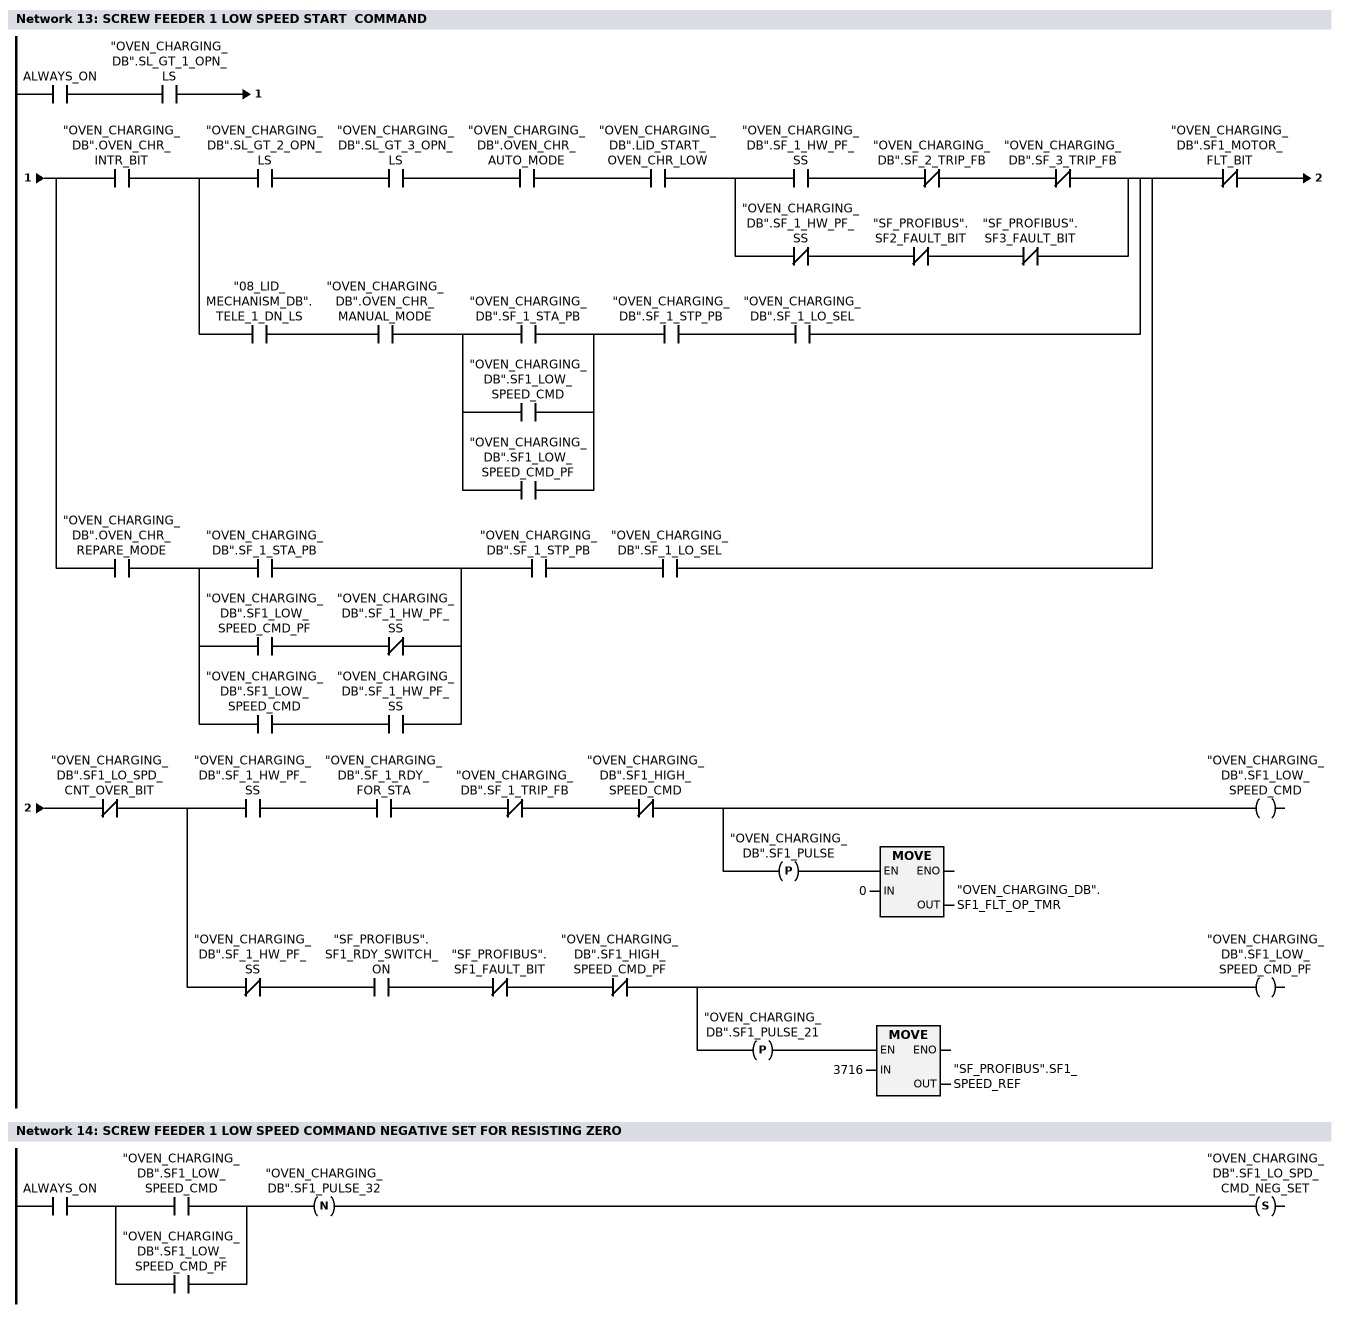
[picture p96: OVEN_CHARGING_SF networks 13-14]
NETWORK
TITLE = SCREW FEEDER 1 LOW SPEED START  COMMAND
      A     "ALWAYS_ON";
      A     "OVEN_CHARGING_DB".SL_GT_1_OPN_LS;
      A(;
      A     "OVEN_CHARGING_DB".OVEN_CHR_INTR_BIT;
      A(;
      A     "OVEN_CHARGING_DB".SL_GT_2_OPN_LS;
      A     "OVEN_CHARGING_DB".SL_GT_3_OPN_LS;
      A     "OVEN_CHARGING_DB".OVEN_CHR_AUTO_MODE;
      A     "OVEN_CHARGING_DB".LID_START_OVEN_CHR_LOW;
      A(;
      A     "OVEN_CHARGING_DB".SF_1_HW_PF_SS;
      AN    "OVEN_CHARGING_DB".SF_2_TRIP_FB;
      AN    "OVEN_CHARGING_DB".SF_3_TRIP_FB;
      O;
      AN    "OVEN_CHARGING_DB".SF_1_HW_PF_SS;
      AN    "SF_PROFIBUS".SF2_FAULT_BIT;
      AN    "SF_PROFIBUS".SF3_FAULT_BIT;
      );
      O;
      A     "08_LID_MECHANISM_DB".TELE_1_DN_LS;
      A     "OVEN_CHARGING_DB".OVEN_CHR_MANUAL_MODE;
      A(;
      O     "OVEN_CHARGING_DB".SF_1_STA_PB;
      O     "OVEN_CHARGING_DB".SF1_LOW_SPEED_CMD;
      O     "OVEN_CHARGING_DB".SF1_LOW_SPEED_CMD_PF;
      );
      A     "OVEN_CHARGING_DB".SF_1_STP_PB;
      A     "OVEN_CHARGING_DB".SF_1_LO_SEL;
      );
      O;
      A     "OVEN_CHARGING_DB".OVEN_CHR_REPARE_MODE;
      A(;
      O     "OVEN_CHARGING_DB".SF_1_STA_PB;
      O;
      A     "OVEN_CHARGING_DB".SF1_LOW_SPEED_CMD_PF;
      AN    "OVEN_CHARGING_DB".SF_1_HW_PF_SS;
      O;
      A     "OVEN_CHARGING_DB".SF1_LOW_SPEED_CMD;
      A     "OVEN_CHARGING_DB".SF_1_HW_PF_SS;
      );
      A     "OVEN_CHARGING_DB".SF_1_STP_PB;
      A     "OVEN_CHARGING_DB".SF_1_LO_SEL;
      );
      AN    "OVEN_CHARGING_DB".SF1_MOTOR_FLT_BIT;
      AN    "OVEN_CHARGING_DB".SF1_LO_SPD_CNT_OVER_BIT;
      =     L 0.0;
      A     L 0.0;
      A     "OVEN_CHARGING_DB".SF_1_HW_PF_SS;
      A     "OVEN_CHARGING_DB".SF_1_RDY_FOR_STA;
      AN    "OVEN_CHARGING_DB".SF_1_TRIP_FB;
      AN    "OVEN_CHARGING_DB".SF1_HIGH_SPEED_CMD;
      =     L 0.1;
      A     L 0.1;
      BLD   102;
      =     "OVEN_CHARGING_DB".SF1_LOW_SPEED_CMD;
      A     L 0.1;
      FP    "OVEN_CHARGING_DB".SF1_PULSE;
      JNB   _007;
      L     0;
      T     "OVEN_CHARGING_DB".SF1_FLT_OP_TMR;
_007: NOP   0;
      A     L 0.0;
      AN    "OVEN_CHARGING_DB".SF_1_HW_PF_SS;
      A     "SF_PROFIBUS".SF1_RDY_SWITCH_ON;
      AN    "SF_PROFIBUS".SF1_FAULT_BIT;
      AN    "OVEN_CHARGING_DB".SF1_HIGH_SPEED_CMD_PF;
      =     L 0.1;
      A     L 0.1;
      BLD   102;
      =     "OVEN_CHARGING_DB".SF1_LOW_SPEED_CMD_PF;
      A     L 0.1;
      FP    "OVEN_CHARGING_DB".SF1_PULSE_21;
      JNB   _008;
      L     3716;
      T     "SF_PROFIBUS".SF1_SPEED_REF;
_008: NOP   0;
NETWORK
TITLE = SCREW FEEDER 1 LOW SPEED COMMAND NEGATIVE SET FOR RESISTING ZERO
      A     "ALWAYS_ON";
      A(;
      O     "OVEN_CHARGING_DB".SF1_LOW_SPEED_CMD;
      O     "OVEN_CHARGING_DB".SF1_LOW_SPEED_CMD_PF;
      );
      FN    "OVEN_CHARGING_DB".SF1_PULSE_32;
      S     "OVEN_CHARGING_DB".SF1_LO_SPD_CMD_NEG_SET;
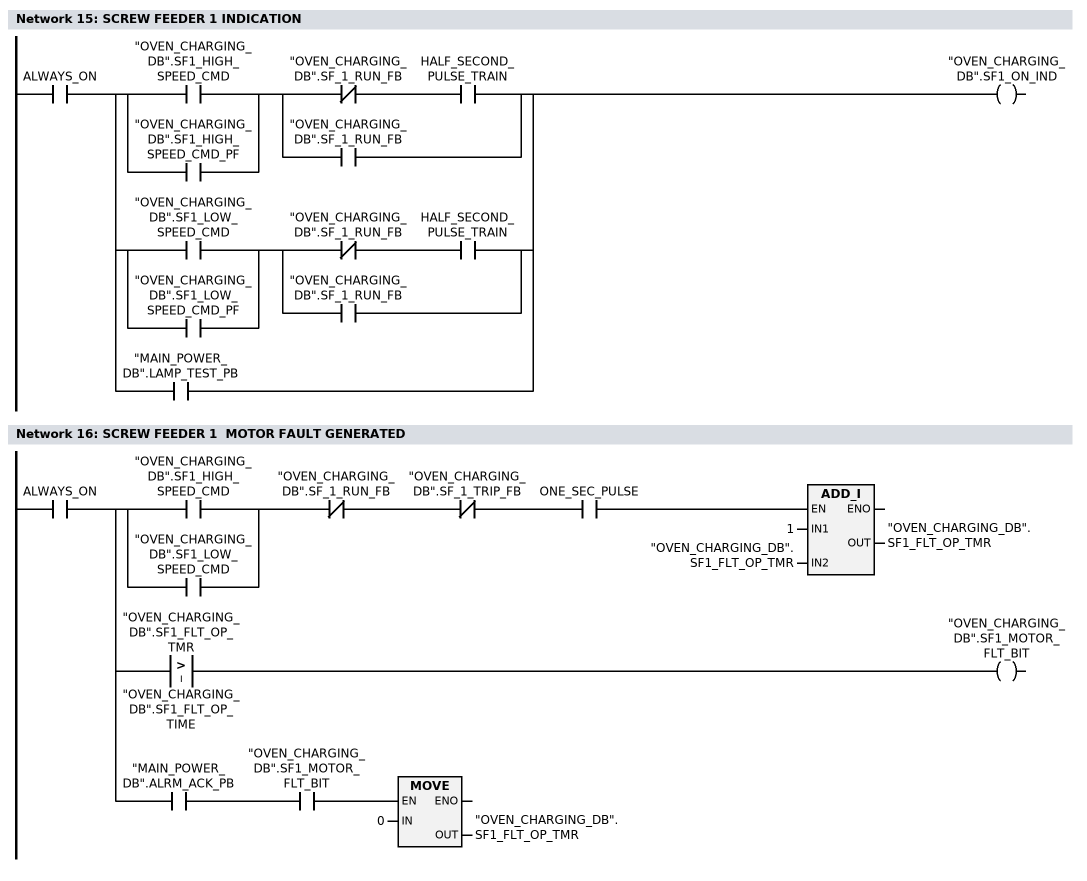
NETWORK
TITLE = SCREW FEEDER 1 INDICATION
      A     "ALWAYS_ON";
      A(;
      A(;
      O     "OVEN_CHARGING_DB".SF1_HIGH_SPEED_CMD;
      O     "OVEN_CHARGING_DB".SF1_HIGH_SPEED_CMD_PF;
      );
      A(;
      AN    "OVEN_CHARGING_DB".SF_1_RUN_FB;
      A     "HALF_SECOND_PULSE_TRAIN";
      O     "OVEN_CHARGING_DB".SF_1_RUN_FB;
      );
      O;
      A(;
      O     "OVEN_CHARGING_DB".SF1_LOW_SPEED_CMD;
      O     "OVEN_CHARGING_DB".SF1_LOW_SPEED_CMD_PF;
      );
      A(;
      AN    "OVEN_CHARGING_DB".SF_1_RUN_FB;
      A     "HALF_SECOND_PULSE_TRAIN";
      O     "OVEN_CHARGING_DB".SF_1_RUN_FB;
      );
      O     "MAIN_POWER_DB".LAMP_TEST_PB;
      );
      =     "OVEN_CHARGING_DB".SF1_ON_IND;
NETWORK
TITLE = SCREW FEEDER 1  MOTOR FAULT GENERATED
      A     "ALWAYS_ON";
      =     L 0.0;
      A     L 0.0;
      A(;
      O     "OVEN_CHARGING_DB".SF1_HIGH_SPEED_CMD;
      O     "OVEN_CHARGING_DB".SF1_LOW_SPEED_CMD;
      );
      AN    "OVEN_CHARGING_DB".SF_1_RUN_FB;
      AN    "OVEN_CHARGING_DB".SF_1_TRIP_FB;
      A     "ONE_SEC_PULSE";
      JNB   _009;
      L     1;
      L     "OVEN_CHARGING_DB".SF1_FLT_OP_TMR;
      +I;
      T     "OVEN_CHARGING_DB".SF1_FLT_OP_TMR;
_009: NOP   0;
      A     L 0.0;
      A(;
      L     "OVEN_CHARGING_DB".SF1_FLT_OP_TMR;
      L     "OVEN_CHARGING_DB".SF1_FLT_OP_TIME;
      >I;
      );
      =     "OVEN_CHARGING_DB".SF1_MOTOR_FLT_BIT;
      A     L 0.0;
      A     "MAIN_POWER_DB".ALRM_ACK_PB;
      A     "OVEN_CHARGING_DB".SF1_MOTOR_FLT_BIT;
      JNB   _00a;
      L     0;
      T     "OVEN_CHARGING_DB".SF1_FLT_OP_TMR;
_00a: NOP   0;
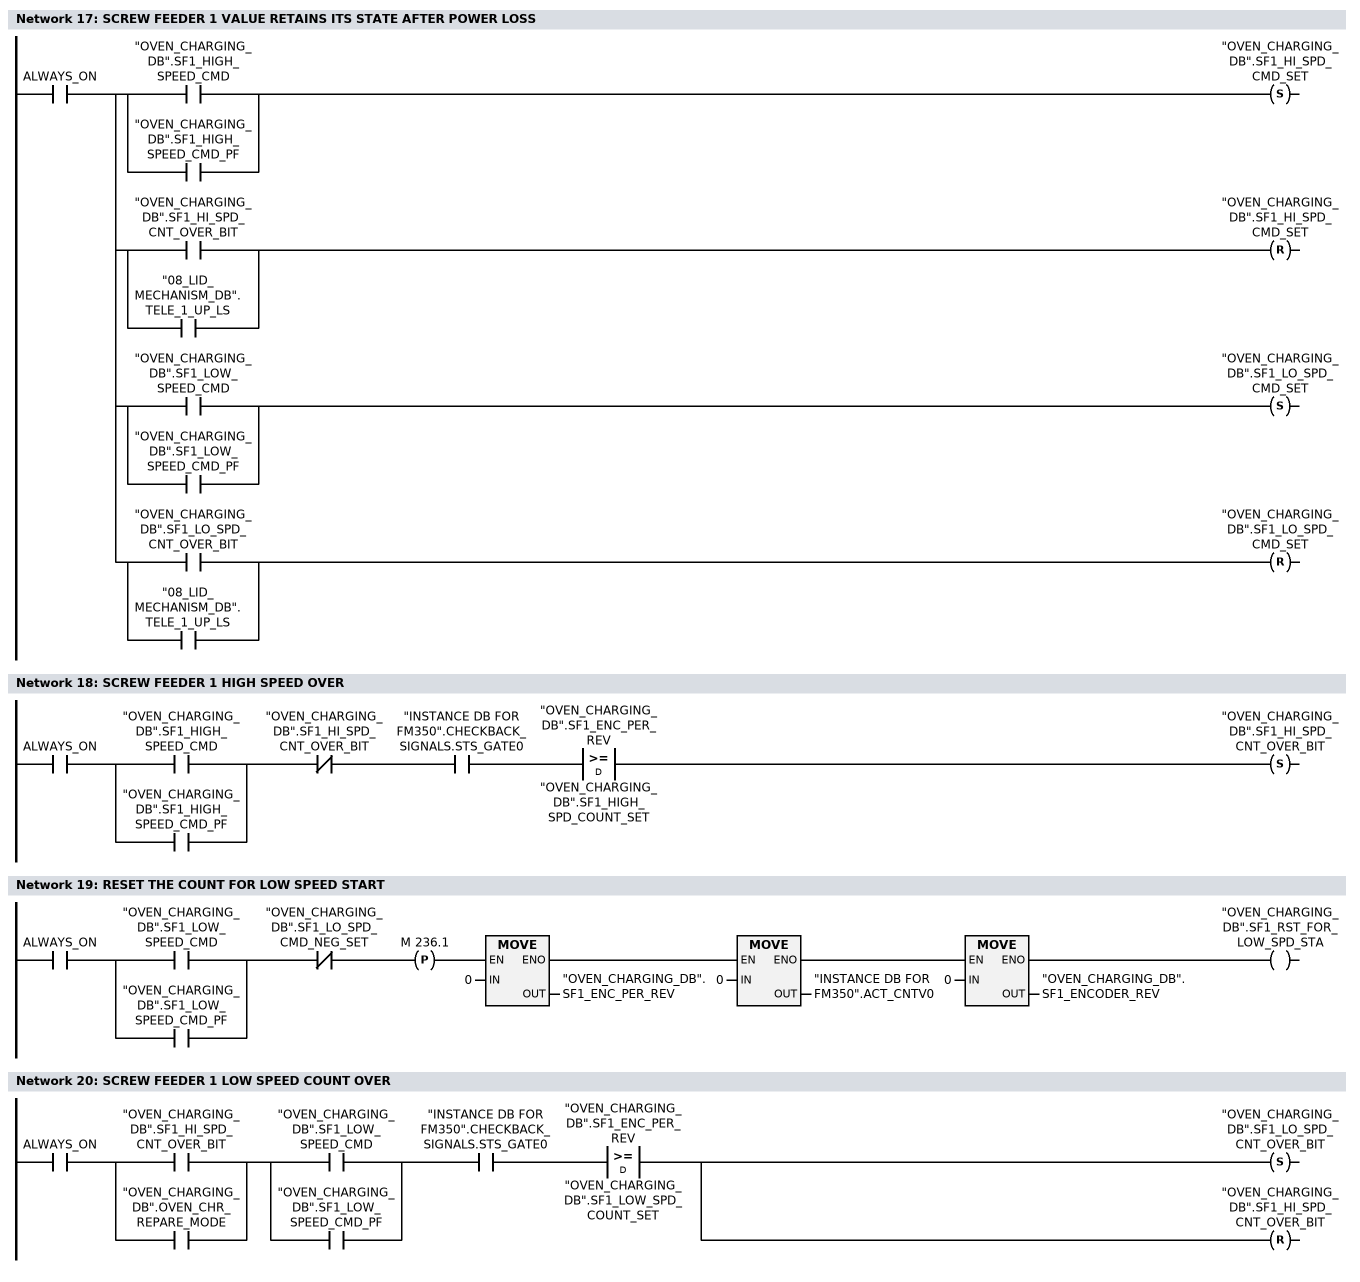
NETWORK
TITLE = SCREW FEEDER 1 VALUE RETAINS ITS STATE AFTER POWER LOSS
      A     "ALWAYS_ON";
      =     L 0.0;
      A     L 0.0;
      A(;
      O     "OVEN_CHARGING_DB".SF1_HIGH_SPEED_CMD;
      O     "OVEN_CHARGING_DB".SF1_HIGH_SPEED_CMD_PF;
      );
      S     "OVEN_CHARGING_DB".SF1_HI_SPD_CMD_SET;
      A     L 0.0;
      A(;
      O     "OVEN_CHARGING_DB".SF1_HI_SPD_CNT_OVER_BIT;
      O     "08_LID_MECHANISM_DB".TELE_1_UP_LS;
      );
      R     "OVEN_CHARGING_DB".SF1_HI_SPD_CMD_SET;
      A     L 0.0;
      A(;
      O     "OVEN_CHARGING_DB".SF1_LOW_SPEED_CMD;
      O     "OVEN_CHARGING_DB".SF1_LOW_SPEED_CMD_PF;
      );
      S     "OVEN_CHARGING_DB".SF1_LO_SPD_CMD_SET;
      A     L 0.0;
      A(;
      O     "OVEN_CHARGING_DB".SF1_LO_SPD_CNT_OVER_BIT;
      O     "08_LID_MECHANISM_DB".TELE_1_UP_LS;
      );
      R     "OVEN_CHARGING_DB".SF1_LO_SPD_CMD_SET;
NETWORK
TITLE = SCREW FEEDER 1 HIGH SPEED OVER
      A     "ALWAYS_ON";
      A(;
      O     "OVEN_CHARGING_DB".SF1_HIGH_SPEED_CMD;
      O     "OVEN_CHARGING_DB".SF1_HIGH_SPEED_CMD_PF;
      );
      AN    "OVEN_CHARGING_DB".SF1_HI_SPD_CNT_OVER_BIT;
      A     "INSTANCE DB FOR FM350".CHECKBACK_SIGNALS.STS_GATE0;
      A(;
      L     "OVEN_CHARGING_DB".SF1_ENC_PER_REV;
      L     "OVEN_CHARGING_DB".SF1_HIGH_SPD_COUNT_SET;
      >=D;
      );
      S     "OVEN_CHARGING_DB".SF1_HI_SPD_CNT_OVER_BIT;
NETWORK
TITLE = RESET THE COUNT FOR LOW SPEED START
      A(;
      A(;
      A     "ALWAYS_ON";
      A(;
      O     "OVEN_CHARGING_DB".SF1_LOW_SPEED_CMD;
      O     "OVEN_CHARGING_DB".SF1_LOW_SPEED_CMD_PF;
      );
      AN    "OVEN_CHARGING_DB".SF1_LO_SPD_CMD_NEG_SET;
      FP    M 236.1;
      JNB   _00b;
      L     0;
      T     "OVEN_CHARGING_DB".SF1_ENC_PER_REV;
      SET;
      SAVE;
      CLR;
_00b: A     BR;
      );
      JNB   _00c;
      L     0;
      T     "INSTANCE DB FOR FM350".ACT_CNTV0;
      SET;
      SAVE;
      CLR;
_00c: A     BR;
      );
      JNB   _00d;
      L     0;
      T     "OVEN_CHARGING_DB".SF1_ENCODER_REV;
      SET;
      SAVE;
      CLR;
_00d: A     BR;
      =     "OVEN_CHARGING_DB".SF1_RST_FOR_LOW_SPD_STA;
NETWORK
TITLE = SCREW FEEDER 1 LOW SPEED COUNT OVER
      A     "ALWAYS_ON";
      A(;
      O     "OVEN_CHARGING_DB".SF1_HI_SPD_CNT_OVER_BIT;
      O     "OVEN_CHARGING_DB".OVEN_CHR_REPARE_MODE;
      );
      A(;
      O     "OVEN_CHARGING_DB".SF1_LOW_SPEED_CMD;
      O     "OVEN_CHARGING_DB".SF1_LOW_SPEED_CMD_PF;
      );
      A     "INSTANCE DB FOR FM350".CHECKBACK_SIGNALS.STS_GATE0;
      A(;
      L     "OVEN_CHARGING_DB".SF1_ENC_PER_REV;
      L     "OVEN_CHARGING_DB".SF1_LOW_SPD_COUNT_SET;
      >=D;
      );
      S     "OVEN_CHARGING_DB".SF1_LO_SPD_CNT_OVER_BIT;
      R     "OVEN_CHARGING_DB".SF1_HI_SPD_CNT_OVER_BIT;
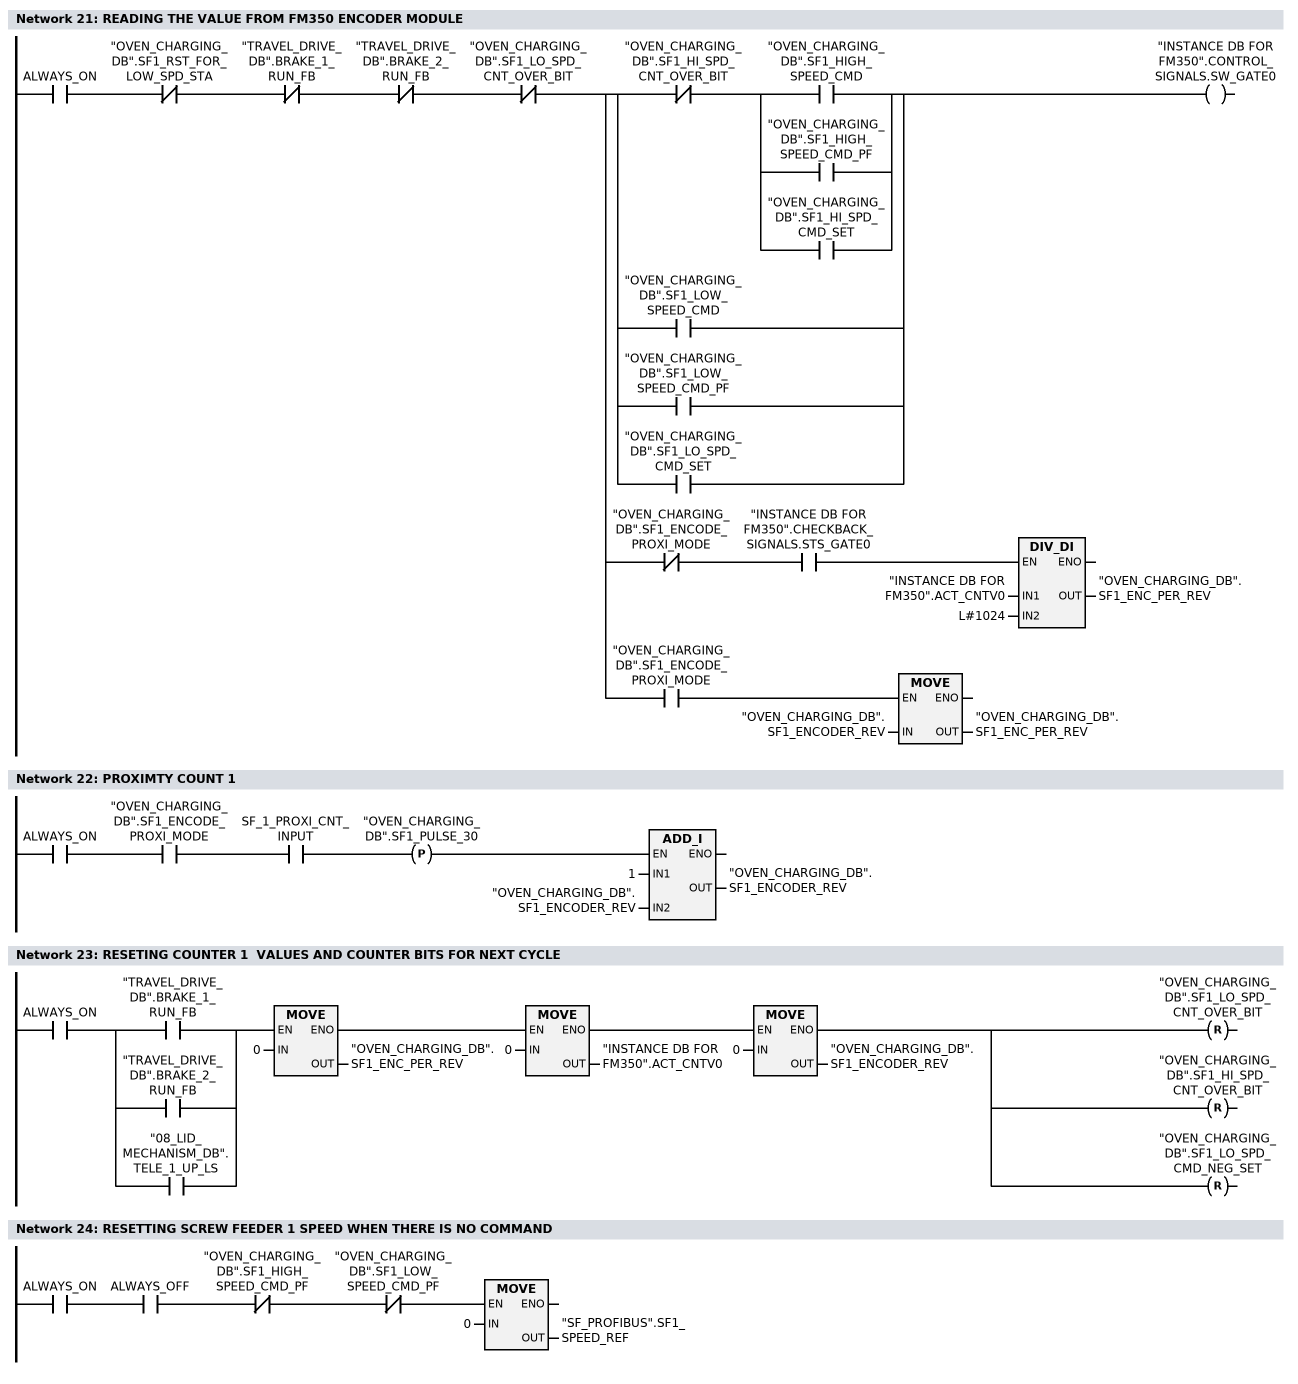
NETWORK
TITLE = READING THE VALUE FROM FM350 ENCODER MODULE 
      A     "ALWAYS_ON";
      AN    "OVEN_CHARGING_DB".SF1_RST_FOR_LOW_SPD_STA;
      AN    "TRAVEL_DRIVE_DB".BRAKE_1_RUN_FB;
      AN    "TRAVEL_DRIVE_DB".BRAKE_2_RUN_FB;
      AN    "OVEN_CHARGING_DB".SF1_LO_SPD_CNT_OVER_BIT;
      =     L 0.0;
      A     L 0.0;
      A(;
      AN    "OVEN_CHARGING_DB".SF1_HI_SPD_CNT_OVER_BIT;
      A(;
      O     "OVEN_CHARGING_DB".SF1_HIGH_SPEED_CMD;
      O     "OVEN_CHARGING_DB".SF1_HIGH_SPEED_CMD_PF;
      O     "OVEN_CHARGING_DB".SF1_HI_SPD_CMD_SET;
      );
      O     "OVEN_CHARGING_DB".SF1_LOW_SPEED_CMD;
      O     "OVEN_CHARGING_DB".SF1_LOW_SPEED_CMD_PF;
      O     "OVEN_CHARGING_DB".SF1_LO_SPD_CMD_SET;
      );
      =     "INSTANCE DB FOR FM350".CONTROL_SIGNALS.SW_GATE0;
      A     L 0.0;
      AN    "OVEN_CHARGING_DB".SF1_ENCODE_PROXI_MODE;
      A     "INSTANCE DB FOR FM350".CHECKBACK_SIGNALS.STS_GATE0;
      JNB   _00e;
      L     "INSTANCE DB FOR FM350".ACT_CNTV0;
      L     L#1024;
      /D;
      T     "OVEN_CHARGING_DB".SF1_ENC_PER_REV;
_00e: NOP   0;
      A     L 0.0;
      A     "OVEN_CHARGING_DB".SF1_ENCODE_PROXI_MODE;
      JNB   _00f;
      L     "OVEN_CHARGING_DB".SF1_ENCODER_REV;
      T     "OVEN_CHARGING_DB".SF1_ENC_PER_REV;
_00f: NOP   0;
NETWORK
TITLE = PROXIMTY COUNT 1
      A     "ALWAYS_ON";
      A     "OVEN_CHARGING_DB".SF1_ENCODE_PROXI_MODE;
      A     "SF_1_PROXI_CNT_INPUT";
      FP    "OVEN_CHARGING_DB".SF1_PULSE_30;
      JNB   _010;
      L     1;
      L     "OVEN_CHARGING_DB".SF1_ENCODER_REV;
      +I;
      T     "OVEN_CHARGING_DB".SF1_ENCODER_REV;
_010: NOP   0;
NETWORK
TITLE = RESETING COUNTER 1  VALUES AND COUNTER BITS FOR NEXT CYCLE
      A(;
      A(;
      A     "ALWAYS_ON";
      A(;
      O     "TRAVEL_DRIVE_DB".BRAKE_1_RUN_FB;
      O     "TRAVEL_DRIVE_DB".BRAKE_2_RUN_FB;
      O     "08_LID_MECHANISM_DB".TELE_1_UP_LS;
      );
      JNB   _011;
      L     0;
      T     "OVEN_CHARGING_DB".SF1_ENC_PER_REV;
      SET;
      SAVE;
      CLR;
_011: A     BR;
      );
      JNB   _012;
      L     0;
      T     "INSTANCE DB FOR FM350".ACT_CNTV0;
      SET;
      SAVE;
      CLR;
_012: A     BR;
      );
      JNB   _013;
      L     0;
      T     "OVEN_CHARGING_DB".SF1_ENCODER_REV;
      SET;
      SAVE;
      CLR;
_013: A     BR;
      R     "OVEN_CHARGING_DB".SF1_LO_SPD_CNT_OVER_BIT;
      R     "OVEN_CHARGING_DB".SF1_HI_SPD_CNT_OVER_BIT;
      R     "OVEN_CHARGING_DB".SF1_LO_SPD_CMD_NEG_SET;
NETWORK
TITLE = RESETTING SCREW FEEDER 1 SPEED WHEN THERE IS NO COMMAND
      A     "ALWAYS_ON";
      A     "ALWAYS_OFF";
      AN    "OVEN_CHARGING_DB".SF1_HIGH_SPEED_CMD_PF;
      AN    "OVEN_CHARGING_DB".SF1_LOW_SPEED_CMD_PF;
      JNB   _014;
      L     0;
      T     "SF_PROFIBUS".SF1_SPEED_REF;
_014: NOP   0;
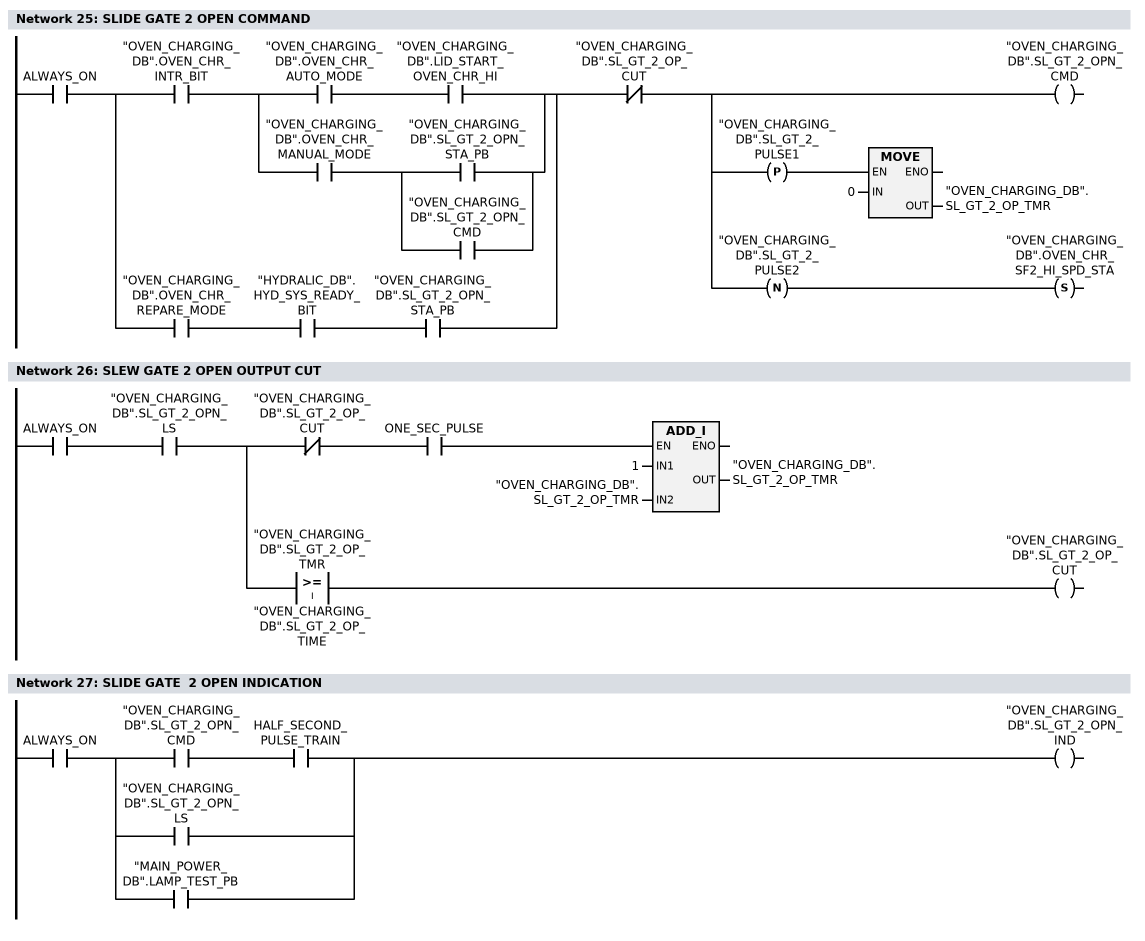
NETWORK
TITLE = SLIDE GATE 2 OPEN COMMAND 
      A     "ALWAYS_ON";
      A(;
      A     "OVEN_CHARGING_DB".OVEN_CHR_INTR_BIT;
      A(;
      A     "OVEN_CHARGING_DB".OVEN_CHR_AUTO_MODE;
      A     "OVEN_CHARGING_DB".LID_START_OVEN_CHR_HI;
      O;
      A     "OVEN_CHARGING_DB".OVEN_CHR_MANUAL_MODE;
      A(;
      O     "OVEN_CHARGING_DB".SL_GT_2_OPN_STA_PB;
      O     "OVEN_CHARGING_DB".SL_GT_2_OPN_CMD;
      );
      );
      O;
      A     "OVEN_CHARGING_DB".OVEN_CHR_REPARE_MODE;
      A     "HYDRALIC_DB".HYD_SYS_READY_BIT;
      A     "OVEN_CHARGING_DB".SL_GT_2_OPN_STA_PB;
      );
      AN    "OVEN_CHARGING_DB".SL_GT_2_OP_CUT;
      =     L 0.0;
      A     L 0.0;
      BLD   102;
      =     "OVEN_CHARGING_DB".SL_GT_2_OPN_CMD;
      A     L 0.0;
      FP    "OVEN_CHARGING_DB".SL_GT_2_PULSE1;
      JNB   _015;
      L     0;
      T     "OVEN_CHARGING_DB".SL_GT_2_OP_TMR;
_015: NOP   0;
      A     L 0.0;
      FN    "OVEN_CHARGING_DB".SL_GT_2_PULSE2;
      S     "OVEN_CHARGING_DB".OVEN_CHR_SF2_HI_SPD_STA;
NETWORK
TITLE = SLEW GATE 2 OPEN OUTPUT CUT
      A     "ALWAYS_ON";
      A     "OVEN_CHARGING_DB".SL_GT_2_OPN_LS;
      =     L 0.0;
      A     L 0.0;
      AN    "OVEN_CHARGING_DB".SL_GT_2_OP_CUT;
      A     "ONE_SEC_PULSE";
      JNB   _016;
      L     1;
      L     "OVEN_CHARGING_DB".SL_GT_2_OP_TMR;
      +I;
      T     "OVEN_CHARGING_DB".SL_GT_2_OP_TMR;
_016: NOP   0;
      A     L 0.0;
      A(;
      L     "OVEN_CHARGING_DB".SL_GT_2_OP_TMR;
      L     "OVEN_CHARGING_DB".SL_GT_2_OP_TIME;
      >=I;
      );
      =     "OVEN_CHARGING_DB".SL_GT_2_OP_CUT;
NETWORK
TITLE = SLIDE GATE  2 OPEN INDICATION
      A     "ALWAYS_ON";
      A(;
      A     "OVEN_CHARGING_DB".SL_GT_2_OPN_CMD;
      A     "HALF_SECOND_PULSE_TRAIN";
      O     "OVEN_CHARGING_DB".SL_GT_2_OPN_LS;
      O     "MAIN_POWER_DB".LAMP_TEST_PB;
      );
      =     "OVEN_CHARGING_DB".SL_GT_2_OPN_IND;
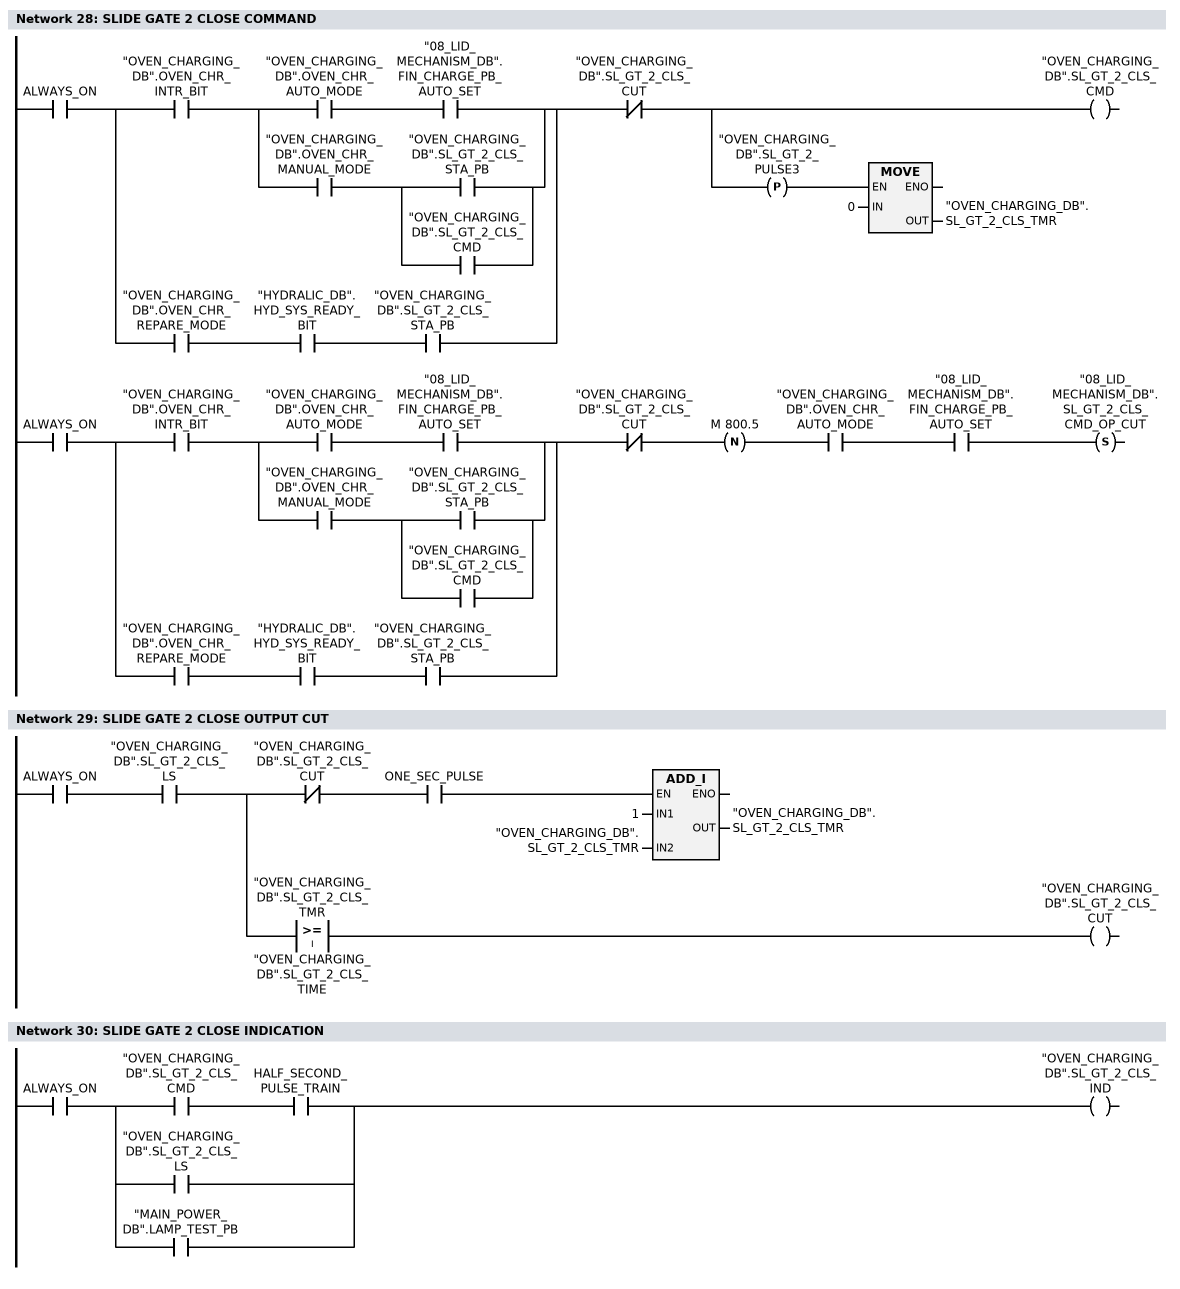
NETWORK
TITLE = SLIDE GATE 2 CLOSE COMMAND
      A     "ALWAYS_ON";
      A(;
      A     "OVEN_CHARGING_DB".OVEN_CHR_INTR_BIT;
      A(;
      A     "OVEN_CHARGING_DB".OVEN_CHR_AUTO_MODE;
      A     "08_LID_MECHANISM_DB".FIN_CHARGE_PB_AUTO_SET;
      O;
      A     "OVEN_CHARGING_DB".OVEN_CHR_MANUAL_MODE;
      A(;
      O     "OVEN_CHARGING_DB".SL_GT_2_CLS_STA_PB;
      O     "OVEN_CHARGING_DB".SL_GT_2_CLS_CMD;
      );
      );
      O;
      A     "OVEN_CHARGING_DB".OVEN_CHR_REPARE_MODE;
      A     "HYDRALIC_DB".HYD_SYS_READY_BIT;
      A     "OVEN_CHARGING_DB".SL_GT_2_CLS_STA_PB;
      );
      AN    "OVEN_CHARGING_DB".SL_GT_2_CLS_CUT;
      =     L 0.0;
      A     L 0.0;
      BLD   102;
      =     "OVEN_CHARGING_DB".SL_GT_2_CLS_CMD;
      A     L 0.0;
      FP    "OVEN_CHARGING_DB".SL_GT_2_PULSE3;
      JNB   _017;
      L     0;
      T     "OVEN_CHARGING_DB".SL_GT_2_CLS_TMR;
_017: NOP   0;
      A(;
      A     L 0.0;
      FN    M 800.5;
      );
      A     "OVEN_CHARGING_DB".OVEN_CHR_AUTO_MODE;
      A     "08_LID_MECHANISM_DB".FIN_CHARGE_PB_AUTO_SET;
      S     "08_LID_MECHANISM_DB".SL_GT_2_CLS_CMD_OP_CUT;
NETWORK
TITLE = SLIDE GATE 2 CLOSE OUTPUT CUT
      A     "ALWAYS_ON";
      A     "OVEN_CHARGING_DB".SL_GT_2_CLS_LS;
      =     L 0.0;
      A     L 0.0;
      AN    "OVEN_CHARGING_DB".SL_GT_2_CLS_CUT;
      A     "ONE_SEC_PULSE";
      JNB   _018;
      L     1;
      L     "OVEN_CHARGING_DB".SL_GT_2_CLS_TMR;
      +I;
      T     "OVEN_CHARGING_DB".SL_GT_2_CLS_TMR;
_018: NOP   0;
      A     L 0.0;
      A(;
      L     "OVEN_CHARGING_DB".SL_GT_2_CLS_TMR;
      L     "OVEN_CHARGING_DB".SL_GT_2_CLS_TIME;
      >=I;
      );
      =     "OVEN_CHARGING_DB".SL_GT_2_CLS_CUT;
NETWORK
TITLE = SLIDE GATE 2 CLOSE INDICATION
      A     "ALWAYS_ON";
      A(;
      A     "OVEN_CHARGING_DB".SL_GT_2_CLS_CMD;
      A     "HALF_SECOND_PULSE_TRAIN";
      O     "OVEN_CHARGING_DB".SL_GT_2_CLS_LS;
      O     "MAIN_POWER_DB".LAMP_TEST_PB;
      );
      =     "OVEN_CHARGING_DB".SL_GT_2_CLS_IND;
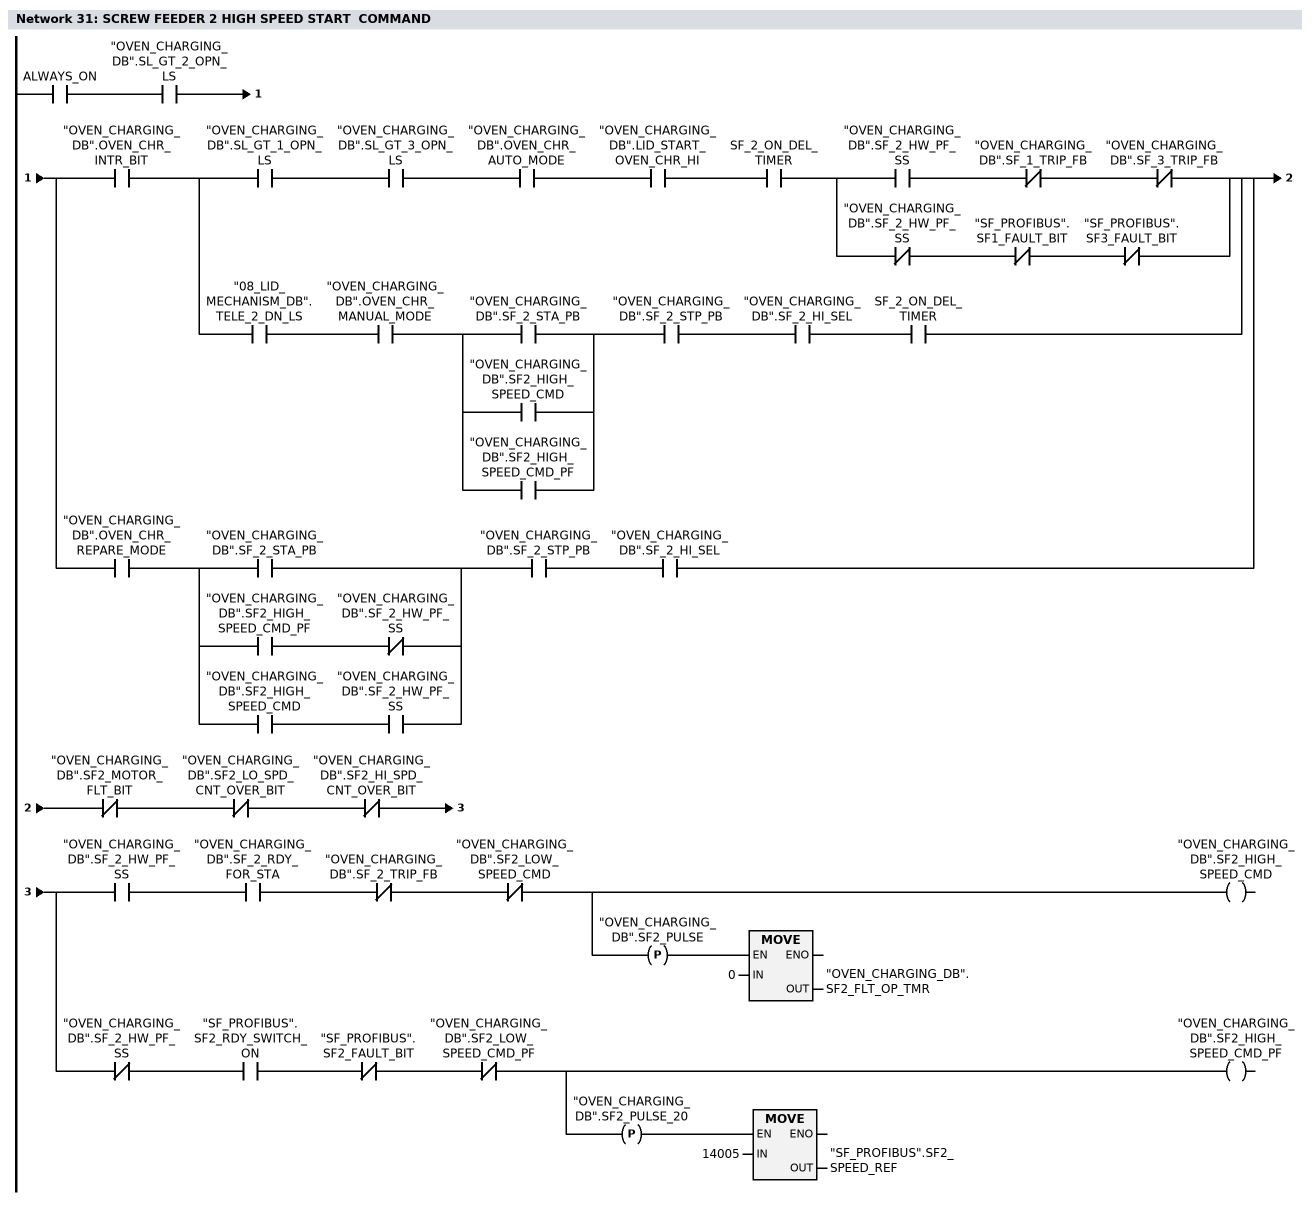
NETWORK
TITLE = SCREW FEEDER 2 HIGH SPEED START  COMMAND
      A     "ALWAYS_ON";
      A     "OVEN_CHARGING_DB".SL_GT_2_OPN_LS;
      A(;
      A     "OVEN_CHARGING_DB".OVEN_CHR_INTR_BIT;
      A(;
      A     "OVEN_CHARGING_DB".SL_GT_1_OPN_LS;
      A     "OVEN_CHARGING_DB".SL_GT_3_OPN_LS;
      A     "OVEN_CHARGING_DB".OVEN_CHR_AUTO_MODE;
      A     "OVEN_CHARGING_DB".LID_START_OVEN_CHR_HI;
      A     "SF_2_ON_DEL_TIMER";
      A(;
      A     "OVEN_CHARGING_DB".SF_2_HW_PF_SS;
      AN    "OVEN_CHARGING_DB".SF_1_TRIP_FB;
      AN    "OVEN_CHARGING_DB".SF_3_TRIP_FB;
      O;
      AN    "OVEN_CHARGING_DB".SF_2_HW_PF_SS;
      AN    "SF_PROFIBUS".SF1_FAULT_BIT;
      AN    "SF_PROFIBUS".SF3_FAULT_BIT;
      );
      O;
      A     "08_LID_MECHANISM_DB".TELE_2_DN_LS;
      A     "OVEN_CHARGING_DB".OVEN_CHR_MANUAL_MODE;
      A(;
      O     "OVEN_CHARGING_DB".SF_2_STA_PB;
      O     "OVEN_CHARGING_DB".SF2_HIGH_SPEED_CMD;
      O     "OVEN_CHARGING_DB".SF2_HIGH_SPEED_CMD_PF;
      );
      A     "OVEN_CHARGING_DB".SF_2_STP_PB;
      A     "OVEN_CHARGING_DB".SF_2_HI_SEL;
      A     "SF_2_ON_DEL_TIMER";
      );
      O;
      A     "OVEN_CHARGING_DB".OVEN_CHR_REPARE_MODE;
      A(;
      O     "OVEN_CHARGING_DB".SF_2_STA_PB;
      O;
      A     "OVEN_CHARGING_DB".SF2_HIGH_SPEED_CMD_PF;
      AN    "OVEN_CHARGING_DB".SF_2_HW_PF_SS;
      O;
      A     "OVEN_CHARGING_DB".SF2_HIGH_SPEED_CMD;
      A     "OVEN_CHARGING_DB".SF_2_HW_PF_SS;
      );
      A     "OVEN_CHARGING_DB".SF_2_STP_PB;
      A     "OVEN_CHARGING_DB".SF_2_HI_SEL;
      );
      AN    "OVEN_CHARGING_DB".SF2_MOTOR_FLT_BIT;
      AN    "OVEN_CHARGING_DB".SF2_LO_SPD_CNT_OVER_BIT;
      AN    "OVEN_CHARGING_DB".SF2_HI_SPD_CNT_OVER_BIT;
      =     L 0.0;
      A     L 0.0;
      A     "OVEN_CHARGING_DB".SF_2_HW_PF_SS;
      A     "OVEN_CHARGING_DB".SF_2_RDY_FOR_STA;
      AN    "OVEN_CHARGING_DB".SF_2_TRIP_FB;
      AN    "OVEN_CHARGING_DB".SF2_LOW_SPEED_CMD;
      =     L 0.1;
      A     L 0.1;
      BLD   102;
      =     "OVEN_CHARGING_DB".SF2_HIGH_SPEED_CMD;
      A     L 0.1;
      FP    "OVEN_CHARGING_DB".SF2_PULSE;
      JNB   _019;
      L     0;
      T     "OVEN_CHARGING_DB".SF2_FLT_OP_TMR;
_019: NOP   0;
      A     L 0.0;
      AN    "OVEN_CHARGING_DB".SF_2_HW_PF_SS;
      A     "SF_PROFIBUS".SF2_RDY_SWITCH_ON;
      AN    "SF_PROFIBUS".SF2_FAULT_BIT;
      AN    "OVEN_CHARGING_DB".SF2_LOW_SPEED_CMD_PF;
      =     L 0.1;
      A     L 0.1;
      BLD   102;
      =     "OVEN_CHARGING_DB".SF2_HIGH_SPEED_CMD_PF;
      A     L 0.1;
      FP    "OVEN_CHARGING_DB".SF2_PULSE_20;
      JNB   _01a;
      L     14005;
      T     "SF_PROFIBUS".SF2_SPEED_REF;
_01a: NOP   0;
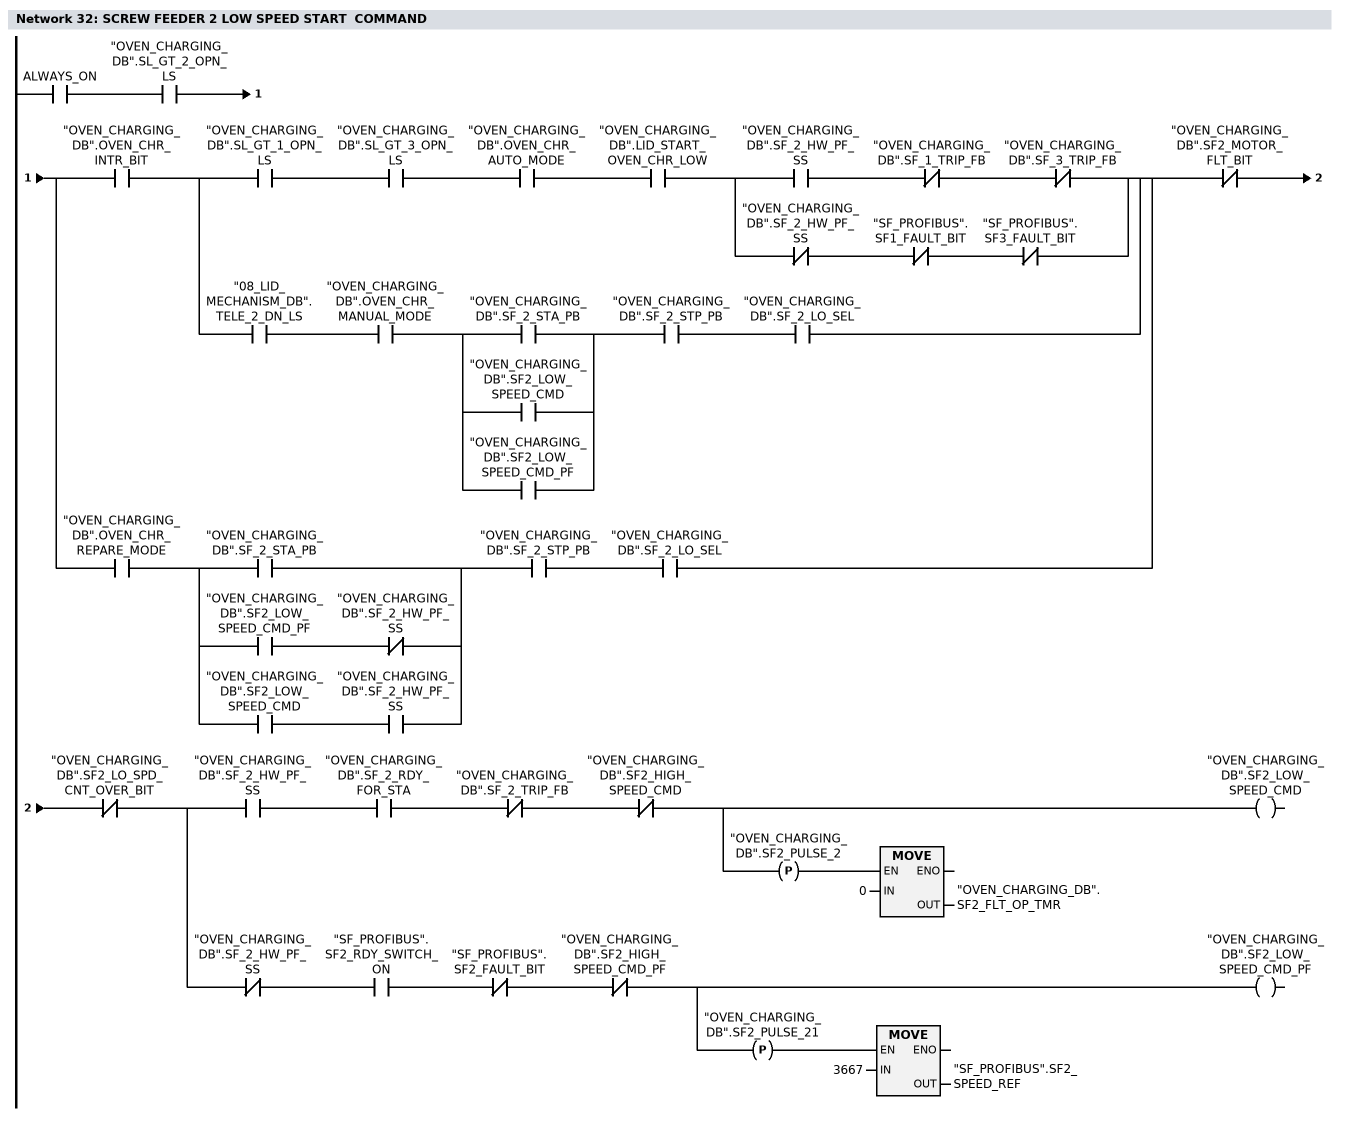
NETWORK
TITLE = SCREW FEEDER 2 LOW SPEED START  COMMAND
      A     "ALWAYS_ON";
      A     "OVEN_CHARGING_DB".SL_GT_2_OPN_LS;
      A(;
      A     "OVEN_CHARGING_DB".OVEN_CHR_INTR_BIT;
      A(;
      A     "OVEN_CHARGING_DB".SL_GT_1_OPN_LS;
      A     "OVEN_CHARGING_DB".SL_GT_3_OPN_LS;
      A     "OVEN_CHARGING_DB".OVEN_CHR_AUTO_MODE;
      A     "OVEN_CHARGING_DB".LID_START_OVEN_CHR_LOW;
      A(;
      A     "OVEN_CHARGING_DB".SF_2_HW_PF_SS;
      AN    "OVEN_CHARGING_DB".SF_1_TRIP_FB;
      AN    "OVEN_CHARGING_DB".SF_3_TRIP_FB;
      O;
      AN    "OVEN_CHARGING_DB".SF_2_HW_PF_SS;
      AN    "SF_PROFIBUS".SF1_FAULT_BIT;
      AN    "SF_PROFIBUS".SF3_FAULT_BIT;
      );
      O;
      A     "08_LID_MECHANISM_DB".TELE_2_DN_LS;
      A     "OVEN_CHARGING_DB".OVEN_CHR_MANUAL_MODE;
      A(;
      O     "OVEN_CHARGING_DB".SF_2_STA_PB;
      O     "OVEN_CHARGING_DB".SF2_LOW_SPEED_CMD;
      O     "OVEN_CHARGING_DB".SF2_LOW_SPEED_CMD_PF;
      );
      A     "OVEN_CHARGING_DB".SF_2_STP_PB;
      A     "OVEN_CHARGING_DB".SF_2_LO_SEL;
      );
      O;
      A     "OVEN_CHARGING_DB".OVEN_CHR_REPARE_MODE;
      A(;
      O     "OVEN_CHARGING_DB".SF_2_STA_PB;
      O;
      A     "OVEN_CHARGING_DB".SF2_LOW_SPEED_CMD_PF;
      AN    "OVEN_CHARGING_DB".SF_2_HW_PF_SS;
      O;
      A     "OVEN_CHARGING_DB".SF2_LOW_SPEED_CMD;
      A     "OVEN_CHARGING_DB".SF_2_HW_PF_SS;
      );
      A     "OVEN_CHARGING_DB".SF_2_STP_PB;
      A     "OVEN_CHARGING_DB".SF_2_LO_SEL;
      );
      AN    "OVEN_CHARGING_DB".SF2_MOTOR_FLT_BIT;
      AN    "OVEN_CHARGING_DB".SF2_LO_SPD_CNT_OVER_BIT;
      =     L 0.0;
      A     L 0.0;
      A     "OVEN_CHARGING_DB".SF_2_HW_PF_SS;
      A     "OVEN_CHARGING_DB".SF_2_RDY_FOR_STA;
      AN    "OVEN_CHARGING_DB".SF_2_TRIP_FB;
      AN    "OVEN_CHARGING_DB".SF2_HIGH_SPEED_CMD;
      =     L 0.1;
      A     L 0.1;
      BLD   102;
      =     "OVEN_CHARGING_DB".SF2_LOW_SPEED_CMD;
      A     L 0.1;
      FP    "OVEN_CHARGING_DB".SF2_PULSE_2;
      JNB   _01b;
      L     0;
      T     "OVEN_CHARGING_DB".SF2_FLT_OP_TMR;
_01b: NOP   0;
      A     L 0.0;
      AN    "OVEN_CHARGING_DB".SF_2_HW_PF_SS;
      A     "SF_PROFIBUS".SF2_RDY_SWITCH_ON;
      AN    "SF_PROFIBUS".SF2_FAULT_BIT;
      AN    "OVEN_CHARGING_DB".SF2_HIGH_SPEED_CMD_PF;
      =     L 0.1;
      A     L 0.1;
      BLD   102;
      =     "OVEN_CHARGING_DB".SF2_LOW_SPEED_CMD_PF;
      A     L 0.1;
      FP    "OVEN_CHARGING_DB".SF2_PULSE_21;
      JNB   _01c;
      L     3667;
      T     "SF_PROFIBUS".SF2_SPEED_REF;
_01c: NOP   0;
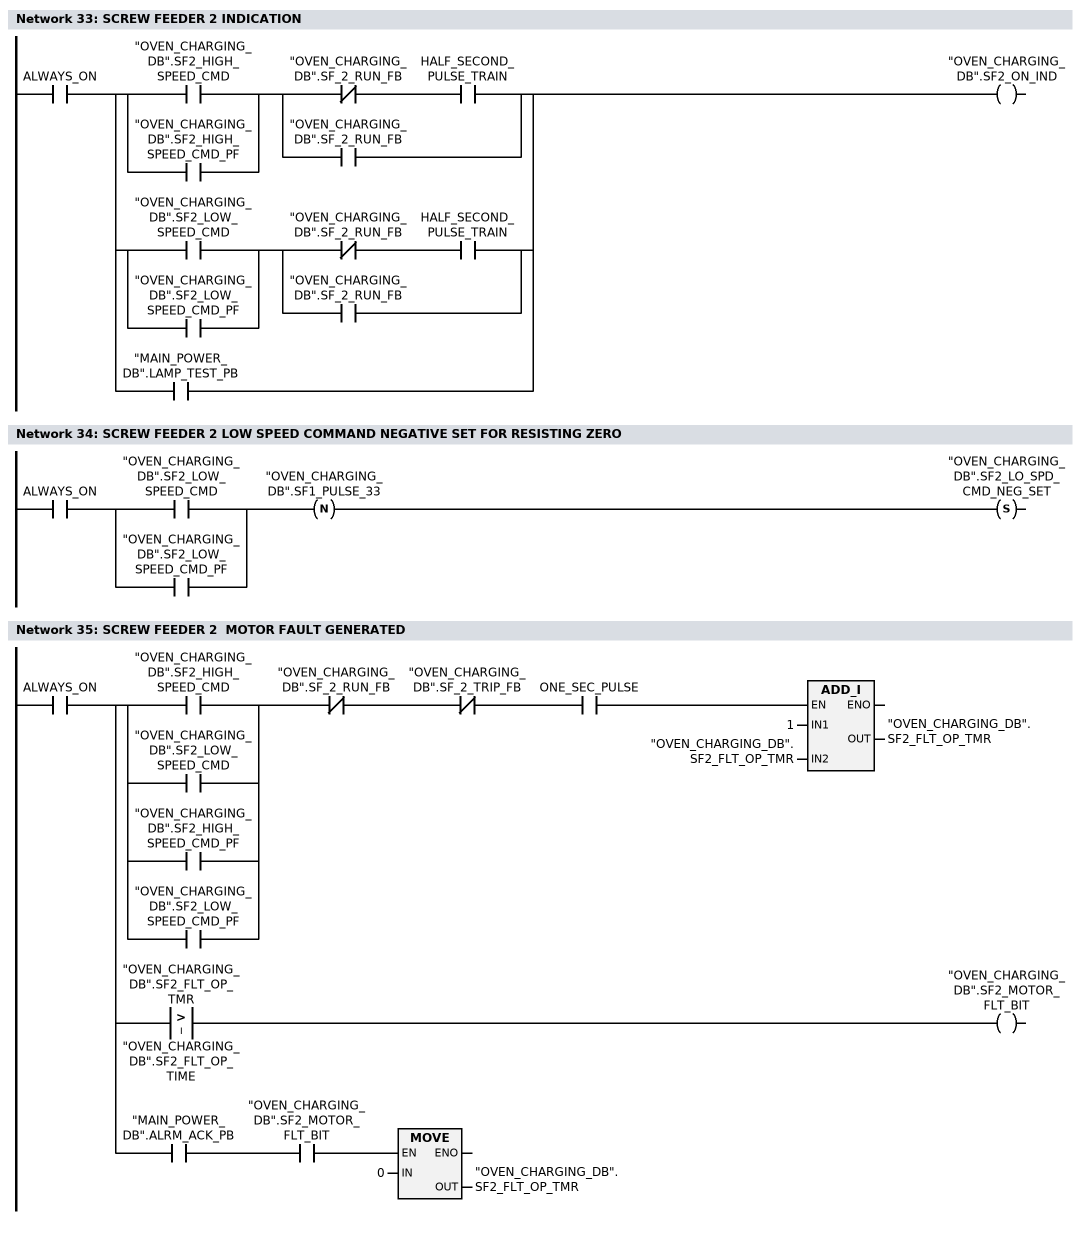
NETWORK
TITLE = SCREW FEEDER 2 INDICATION
      A     "ALWAYS_ON";
      A(;
      A(;
      O     "OVEN_CHARGING_DB".SF2_HIGH_SPEED_CMD;
      O     "OVEN_CHARGING_DB".SF2_HIGH_SPEED_CMD_PF;
      );
      A(;
      AN    "OVEN_CHARGING_DB".SF_2_RUN_FB;
      A     "HALF_SECOND_PULSE_TRAIN";
      O     "OVEN_CHARGING_DB".SF_2_RUN_FB;
      );
      O;
      A(;
      O     "OVEN_CHARGING_DB".SF2_LOW_SPEED_CMD;
      O     "OVEN_CHARGING_DB".SF2_LOW_SPEED_CMD_PF;
      );
      A(;
      AN    "OVEN_CHARGING_DB".SF_2_RUN_FB;
      A     "HALF_SECOND_PULSE_TRAIN";
      O     "OVEN_CHARGING_DB".SF_2_RUN_FB;
      );
      O     "MAIN_POWER_DB".LAMP_TEST_PB;
      );
      =     "OVEN_CHARGING_DB".SF2_ON_IND;
NETWORK
TITLE = SCREW FEEDER 2 LOW SPEED COMMAND NEGATIVE SET FOR RESISTING ZERO
      A     "ALWAYS_ON";
      A(;
      O     "OVEN_CHARGING_DB".SF2_LOW_SPEED_CMD;
      O     "OVEN_CHARGING_DB".SF2_LOW_SPEED_CMD_PF;
      );
      FN    "OVEN_CHARGING_DB".SF1_PULSE_33;
      S     "OVEN_CHARGING_DB".SF2_LO_SPD_CMD_NEG_SET;
NETWORK
TITLE = SCREW FEEDER 2  MOTOR FAULT GENERATED
      A     "ALWAYS_ON";
      =     L 0.0;
      A     L 0.0;
      A(;
      O     "OVEN_CHARGING_DB".SF2_HIGH_SPEED_CMD;
      O     "OVEN_CHARGING_DB".SF2_LOW_SPEED_CMD;
      O     "OVEN_CHARGING_DB".SF2_HIGH_SPEED_CMD_PF;
      O     "OVEN_CHARGING_DB".SF2_LOW_SPEED_CMD_PF;
      );
      AN    "OVEN_CHARGING_DB".SF_2_RUN_FB;
      AN    "OVEN_CHARGING_DB".SF_2_TRIP_FB;
      A     "ONE_SEC_PULSE";
      JNB   _01d;
      L     1;
      L     "OVEN_CHARGING_DB".SF2_FLT_OP_TMR;
      +I;
      T     "OVEN_CHARGING_DB".SF2_FLT_OP_TMR;
_01d: NOP   0;
      A     L 0.0;
      A(;
      L     "OVEN_CHARGING_DB".SF2_FLT_OP_TMR;
      L     "OVEN_CHARGING_DB".SF2_FLT_OP_TIME;
      >I;
      );
      =     "OVEN_CHARGING_DB".SF2_MOTOR_FLT_BIT;
      A     L 0.0;
      A     "MAIN_POWER_DB".ALRM_ACK_PB;
      A     "OVEN_CHARGING_DB".SF2_MOTOR_FLT_BIT;
      JNB   _01e;
      L     0;
      T     "OVEN_CHARGING_DB".SF2_FLT_OP_TMR;
_01e: NOP   0;
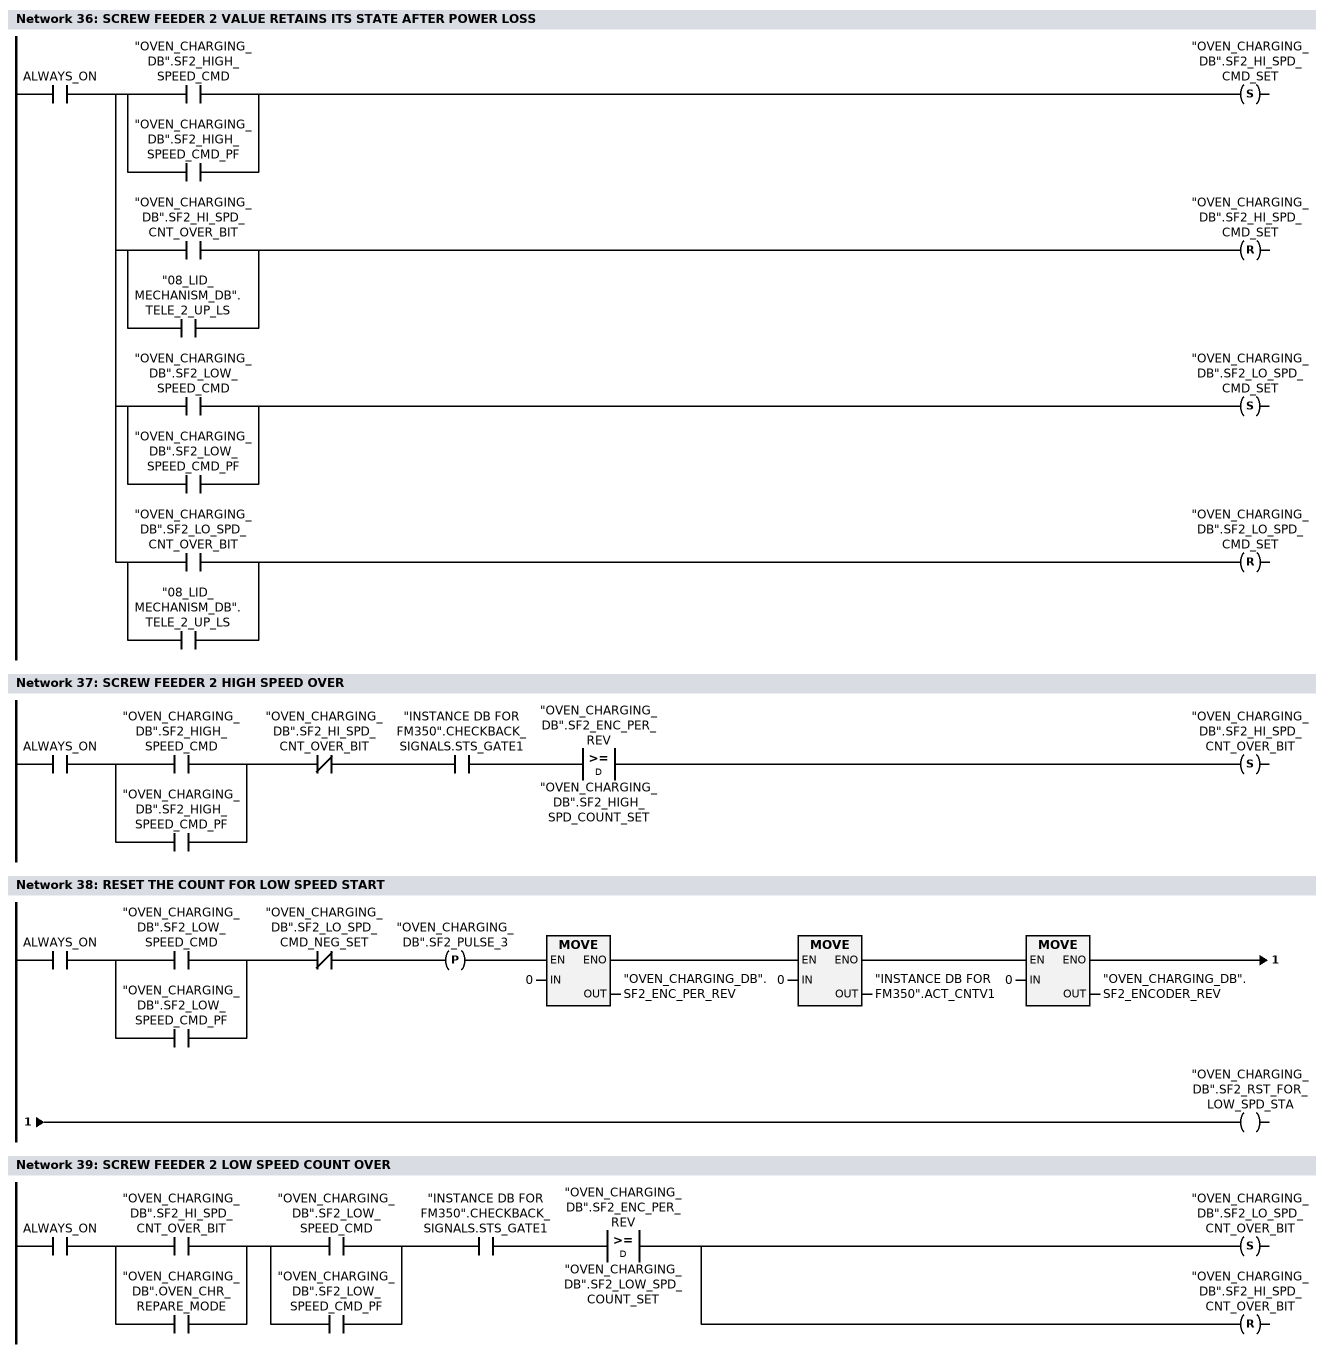
NETWORK
TITLE = SCREW FEEDER 2 VALUE RETAINS ITS STATE AFTER POWER LOSS
      A     "ALWAYS_ON";
      =     L 0.0;
      A     L 0.0;
      A(;
      O     "OVEN_CHARGING_DB".SF2_HIGH_SPEED_CMD;
      O     "OVEN_CHARGING_DB".SF2_HIGH_SPEED_CMD_PF;
      );
      S     "OVEN_CHARGING_DB".SF2_HI_SPD_CMD_SET;
      A     L 0.0;
      A(;
      O     "OVEN_CHARGING_DB".SF2_HI_SPD_CNT_OVER_BIT;
      O     "08_LID_MECHANISM_DB".TELE_2_UP_LS;
      );
      R     "OVEN_CHARGING_DB".SF2_HI_SPD_CMD_SET;
      A     L 0.0;
      A(;
      O     "OVEN_CHARGING_DB".SF2_LOW_SPEED_CMD;
      O     "OVEN_CHARGING_DB".SF2_LOW_SPEED_CMD_PF;
      );
      S     "OVEN_CHARGING_DB".SF2_LO_SPD_CMD_SET;
      A     L 0.0;
      A(;
      O     "OVEN_CHARGING_DB".SF2_LO_SPD_CNT_OVER_BIT;
      O     "08_LID_MECHANISM_DB".TELE_2_UP_LS;
      );
      R     "OVEN_CHARGING_DB".SF2_LO_SPD_CMD_SET;
NETWORK
TITLE = SCREW FEEDER 2 HIGH SPEED OVER
      A     "ALWAYS_ON";
      A(;
      O     "OVEN_CHARGING_DB".SF2_HIGH_SPEED_CMD;
      O     "OVEN_CHARGING_DB".SF2_HIGH_SPEED_CMD_PF;
      );
      AN    "OVEN_CHARGING_DB".SF2_HI_SPD_CNT_OVER_BIT;
      A     "INSTANCE DB FOR FM350".CHECKBACK_SIGNALS.STS_GATE1;
      A(;
      L     "OVEN_CHARGING_DB".SF2_ENC_PER_REV;
      L     "OVEN_CHARGING_DB".SF2_HIGH_SPD_COUNT_SET;
      >=D;
      );
      S     "OVEN_CHARGING_DB".SF2_HI_SPD_CNT_OVER_BIT;
NETWORK
TITLE = RESET THE COUNT FOR LOW SPEED START
      A(;
      A(;
      A     "ALWAYS_ON";
      A(;
      O     "OVEN_CHARGING_DB".SF2_LOW_SPEED_CMD;
      O     "OVEN_CHARGING_DB".SF2_LOW_SPEED_CMD_PF;
      );
      AN    "OVEN_CHARGING_DB".SF2_LO_SPD_CMD_NEG_SET;
      FP    "OVEN_CHARGING_DB".SF2_PULSE_3;
      JNB   _01f;
      L     0;
      T     "OVEN_CHARGING_DB".SF2_ENC_PER_REV;
      SET;
      SAVE;
      CLR;
_01f: A     BR;
      );
      JNB   _020;
      L     0;
      T     "INSTANCE DB FOR FM350".ACT_CNTV1;
      SET;
      SAVE;
      CLR;
_020: A     BR;
      );
      JNB   _021;
      L     0;
      T     "OVEN_CHARGING_DB".SF2_ENCODER_REV;
      SET;
      SAVE;
      CLR;
_021: A     BR;
      =     "OVEN_CHARGING_DB".SF2_RST_FOR_LOW_SPD_STA;
NETWORK
TITLE = SCREW FEEDER 2 LOW SPEED COUNT OVER
      A     "ALWAYS_ON";
      A(;
      O     "OVEN_CHARGING_DB".SF2_HI_SPD_CNT_OVER_BIT;
      O     "OVEN_CHARGING_DB".OVEN_CHR_REPARE_MODE;
      );
      A(;
      O     "OVEN_CHARGING_DB".SF2_LOW_SPEED_CMD;
      O     "OVEN_CHARGING_DB".SF2_LOW_SPEED_CMD_PF;
      );
      A     "INSTANCE DB FOR FM350".CHECKBACK_SIGNALS.STS_GATE1;
      A(;
      L     "OVEN_CHARGING_DB".SF2_ENC_PER_REV;
      L     "OVEN_CHARGING_DB".SF2_LOW_SPD_COUNT_SET;
      >=D;
      );
      S     "OVEN_CHARGING_DB".SF2_LO_SPD_CNT_OVER_BIT;
      R     "OVEN_CHARGING_DB".SF2_HI_SPD_CNT_OVER_BIT;
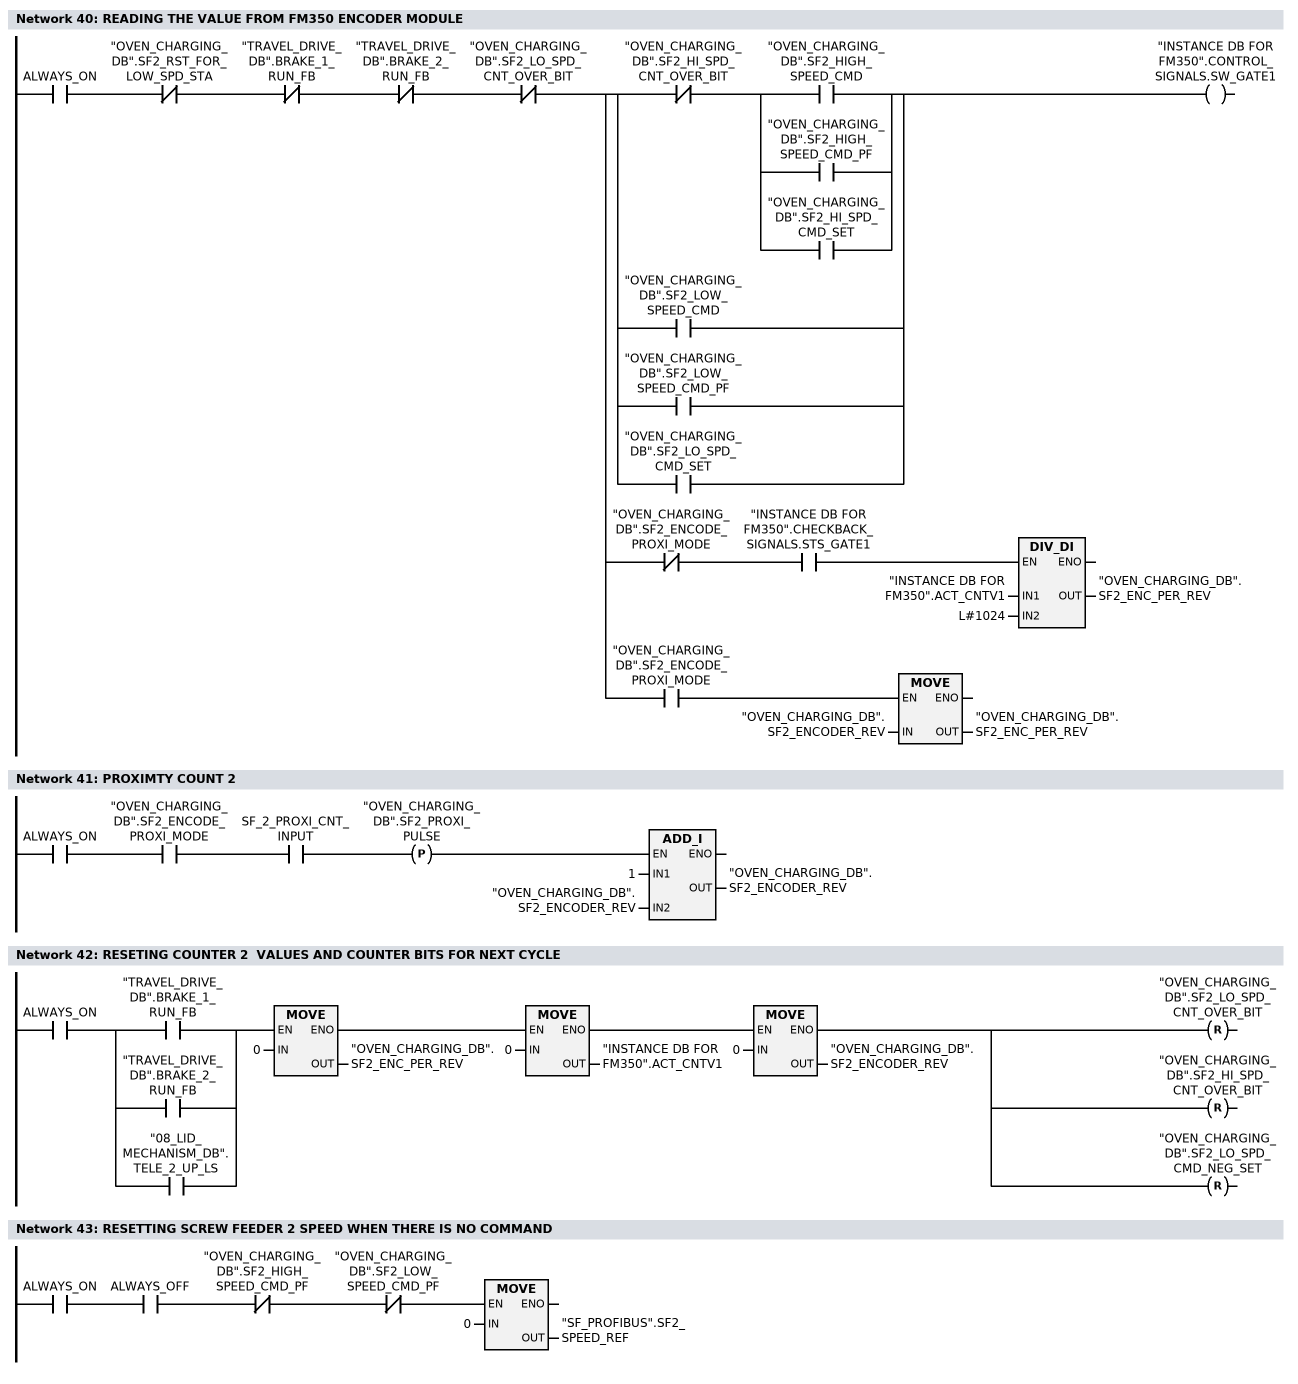
NETWORK
TITLE = READING THE VALUE FROM FM350 ENCODER MODULE 
//FOR SECOND SCREW FEEDER 
      A     "ALWAYS_ON";
      AN    "OVEN_CHARGING_DB".SF2_RST_FOR_LOW_SPD_STA;
      AN    "TRAVEL_DRIVE_DB".BRAKE_1_RUN_FB;
      AN    "TRAVEL_DRIVE_DB".BRAKE_2_RUN_FB;
      AN    "OVEN_CHARGING_DB".SF2_LO_SPD_CNT_OVER_BIT;
      =     L 0.0;
      A     L 0.0;
      A(;
      AN    "OVEN_CHARGING_DB".SF2_HI_SPD_CNT_OVER_BIT;
      A(;
      O     "OVEN_CHARGING_DB".SF2_HIGH_SPEED_CMD;
      O     "OVEN_CHARGING_DB".SF2_HIGH_SPEED_CMD_PF;
      O     "OVEN_CHARGING_DB".SF2_HI_SPD_CMD_SET;
      );
      O     "OVEN_CHARGING_DB".SF2_LOW_SPEED_CMD;
      O     "OVEN_CHARGING_DB".SF2_LOW_SPEED_CMD_PF;
      O     "OVEN_CHARGING_DB".SF2_LO_SPD_CMD_SET;
      );
      =     "INSTANCE DB FOR FM350".CONTROL_SIGNALS.SW_GATE1;
      A     L 0.0;
      AN    "OVEN_CHARGING_DB".SF2_ENCODE_PROXI_MODE;
      A     "INSTANCE DB FOR FM350".CHECKBACK_SIGNALS.STS_GATE1;
      JNB   _022;
      L     "INSTANCE DB FOR FM350".ACT_CNTV1;
      L     L#1024;
      /D;
      T     "OVEN_CHARGING_DB".SF2_ENC_PER_REV;
_022: NOP   0;
      A     L 0.0;
      A     "OVEN_CHARGING_DB".SF2_ENCODE_PROXI_MODE;
      JNB   _023;
      L     "OVEN_CHARGING_DB".SF2_ENCODER_REV;
      T     "OVEN_CHARGING_DB".SF2_ENC_PER_REV;
_023: NOP   0;
NETWORK
TITLE = PROXIMTY COUNT 2
      A     "ALWAYS_ON";
      A     "OVEN_CHARGING_DB".SF2_ENCODE_PROXI_MODE;
      A     "SF_2_PROXI_CNT_INPUT";
      FP    "OVEN_CHARGING_DB".SF2_PROXI_PULSE;
      JNB   _024;
      L     1;
      L     "OVEN_CHARGING_DB".SF2_ENCODER_REV;
      +I;
      T     "OVEN_CHARGING_DB".SF2_ENCODER_REV;
_024: NOP   0;
NETWORK
TITLE = RESETING COUNTER 2  VALUES AND COUNTER BITS FOR NEXT CYCLE
      A(;
      A(;
      A     "ALWAYS_ON";
      A(;
      O     "TRAVEL_DRIVE_DB".BRAKE_1_RUN_FB;
      O     "TRAVEL_DRIVE_DB".BRAKE_2_RUN_FB;
      O     "08_LID_MECHANISM_DB".TELE_2_UP_LS;
      );
      JNB   _025;
      L     0;
      T     "OVEN_CHARGING_DB".SF2_ENC_PER_REV;
      SET;
      SAVE;
      CLR;
_025: A     BR;
      );
      JNB   _026;
      L     0;
      T     "INSTANCE DB FOR FM350".ACT_CNTV1;
      SET;
      SAVE;
      CLR;
_026: A     BR;
      );
      JNB   _027;
      L     0;
      T     "OVEN_CHARGING_DB".SF2_ENCODER_REV;
      SET;
      SAVE;
      CLR;
_027: A     BR;
      R     "OVEN_CHARGING_DB".SF2_LO_SPD_CNT_OVER_BIT;
      R     "OVEN_CHARGING_DB".SF2_HI_SPD_CNT_OVER_BIT;
      R     "OVEN_CHARGING_DB".SF2_LO_SPD_CMD_NEG_SET;
NETWORK
TITLE = RESETTING SCREW FEEDER 2 SPEED WHEN THERE IS NO COMMAND
      A     "ALWAYS_ON";
      A     "ALWAYS_OFF";
      AN    "OVEN_CHARGING_DB".SF2_HIGH_SPEED_CMD_PF;
      AN    "OVEN_CHARGING_DB".SF2_LOW_SPEED_CMD_PF;
      JNB   _028;
      L     0;
      T     "SF_PROFIBUS".SF2_SPEED_REF;
_028: NOP   0;
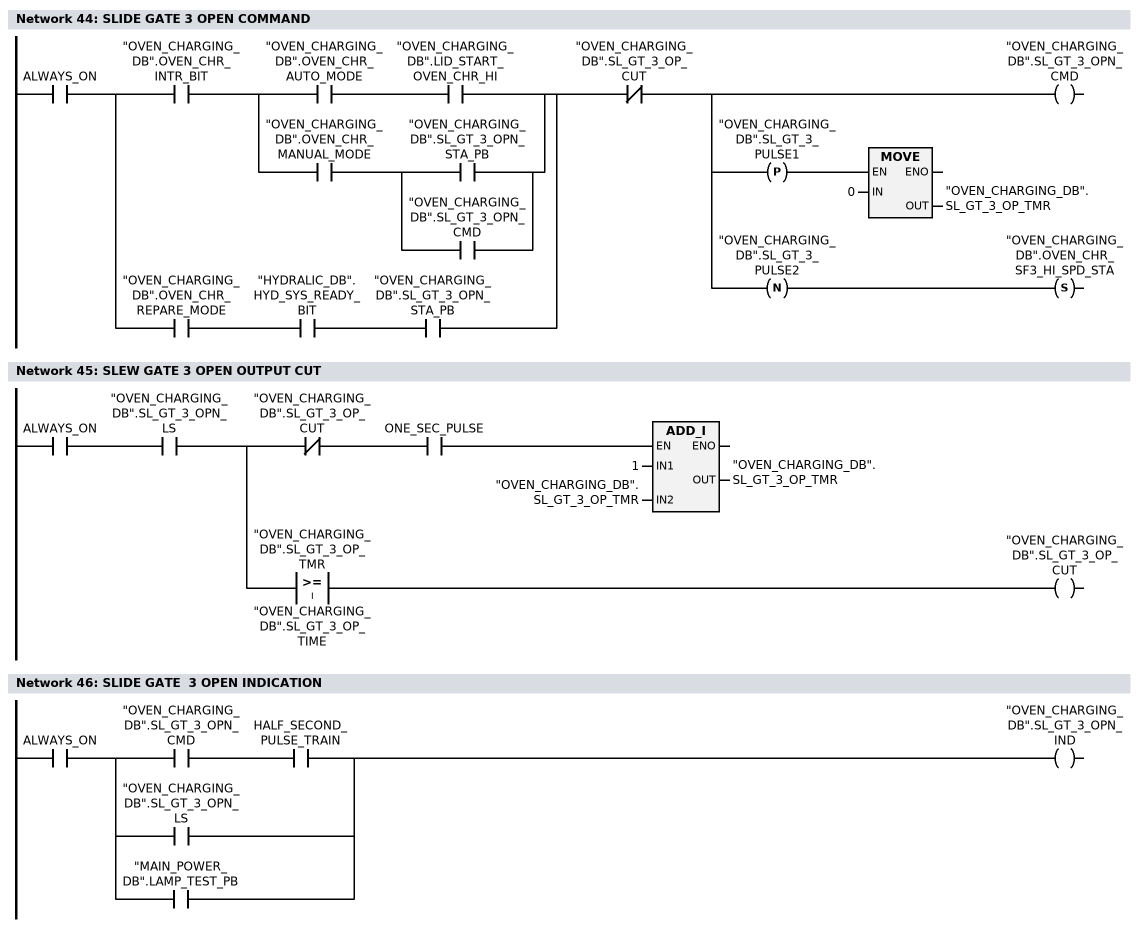
NETWORK
TITLE = SLIDE GATE 3 OPEN COMMAND 
      A     "ALWAYS_ON";
      A(;
      A     "OVEN_CHARGING_DB".OVEN_CHR_INTR_BIT;
      A(;
      A     "OVEN_CHARGING_DB".OVEN_CHR_AUTO_MODE;
      A     "OVEN_CHARGING_DB".LID_START_OVEN_CHR_HI;
      O;
      A     "OVEN_CHARGING_DB".OVEN_CHR_MANUAL_MODE;
      A(;
      O     "OVEN_CHARGING_DB".SL_GT_3_OPN_STA_PB;
      O     "OVEN_CHARGING_DB".SL_GT_3_OPN_CMD;
      );
      );
      O;
      A     "OVEN_CHARGING_DB".OVEN_CHR_REPARE_MODE;
      A     "HYDRALIC_DB".HYD_SYS_READY_BIT;
      A     "OVEN_CHARGING_DB".SL_GT_3_OPN_STA_PB;
      );
      AN    "OVEN_CHARGING_DB".SL_GT_3_OP_CUT;
      =     L 0.0;
      A     L 0.0;
      BLD   102;
      =     "OVEN_CHARGING_DB".SL_GT_3_OPN_CMD;
      A     L 0.0;
      FP    "OVEN_CHARGING_DB".SL_GT_3_PULSE1;
      JNB   _029;
      L     0;
      T     "OVEN_CHARGING_DB".SL_GT_3_OP_TMR;
_029: NOP   0;
      A     L 0.0;
      FN    "OVEN_CHARGING_DB".SL_GT_3_PULSE2;
      S     "OVEN_CHARGING_DB".OVEN_CHR_SF3_HI_SPD_STA;
NETWORK
TITLE = SLEW GATE 3 OPEN OUTPUT CUT
      A     "ALWAYS_ON";
      A     "OVEN_CHARGING_DB".SL_GT_3_OPN_LS;
      =     L 0.0;
      A     L 0.0;
      AN    "OVEN_CHARGING_DB".SL_GT_3_OP_CUT;
      A     "ONE_SEC_PULSE";
      JNB   _02a;
      L     1;
      L     "OVEN_CHARGING_DB".SL_GT_3_OP_TMR;
      +I;
      T     "OVEN_CHARGING_DB".SL_GT_3_OP_TMR;
_02a: NOP   0;
      A     L 0.0;
      A(;
      L     "OVEN_CHARGING_DB".SL_GT_3_OP_TMR;
      L     "OVEN_CHARGING_DB".SL_GT_3_OP_TIME;
      >=I;
      );
      =     "OVEN_CHARGING_DB".SL_GT_3_OP_CUT;
NETWORK
TITLE = SLIDE GATE  3 OPEN INDICATION
      A     "ALWAYS_ON";
      A(;
      A     "OVEN_CHARGING_DB".SL_GT_3_OPN_CMD;
      A     "HALF_SECOND_PULSE_TRAIN";
      O     "OVEN_CHARGING_DB".SL_GT_3_OPN_LS;
      O     "MAIN_POWER_DB".LAMP_TEST_PB;
      );
      =     "OVEN_CHARGING_DB".SL_GT_3_OPN_IND;
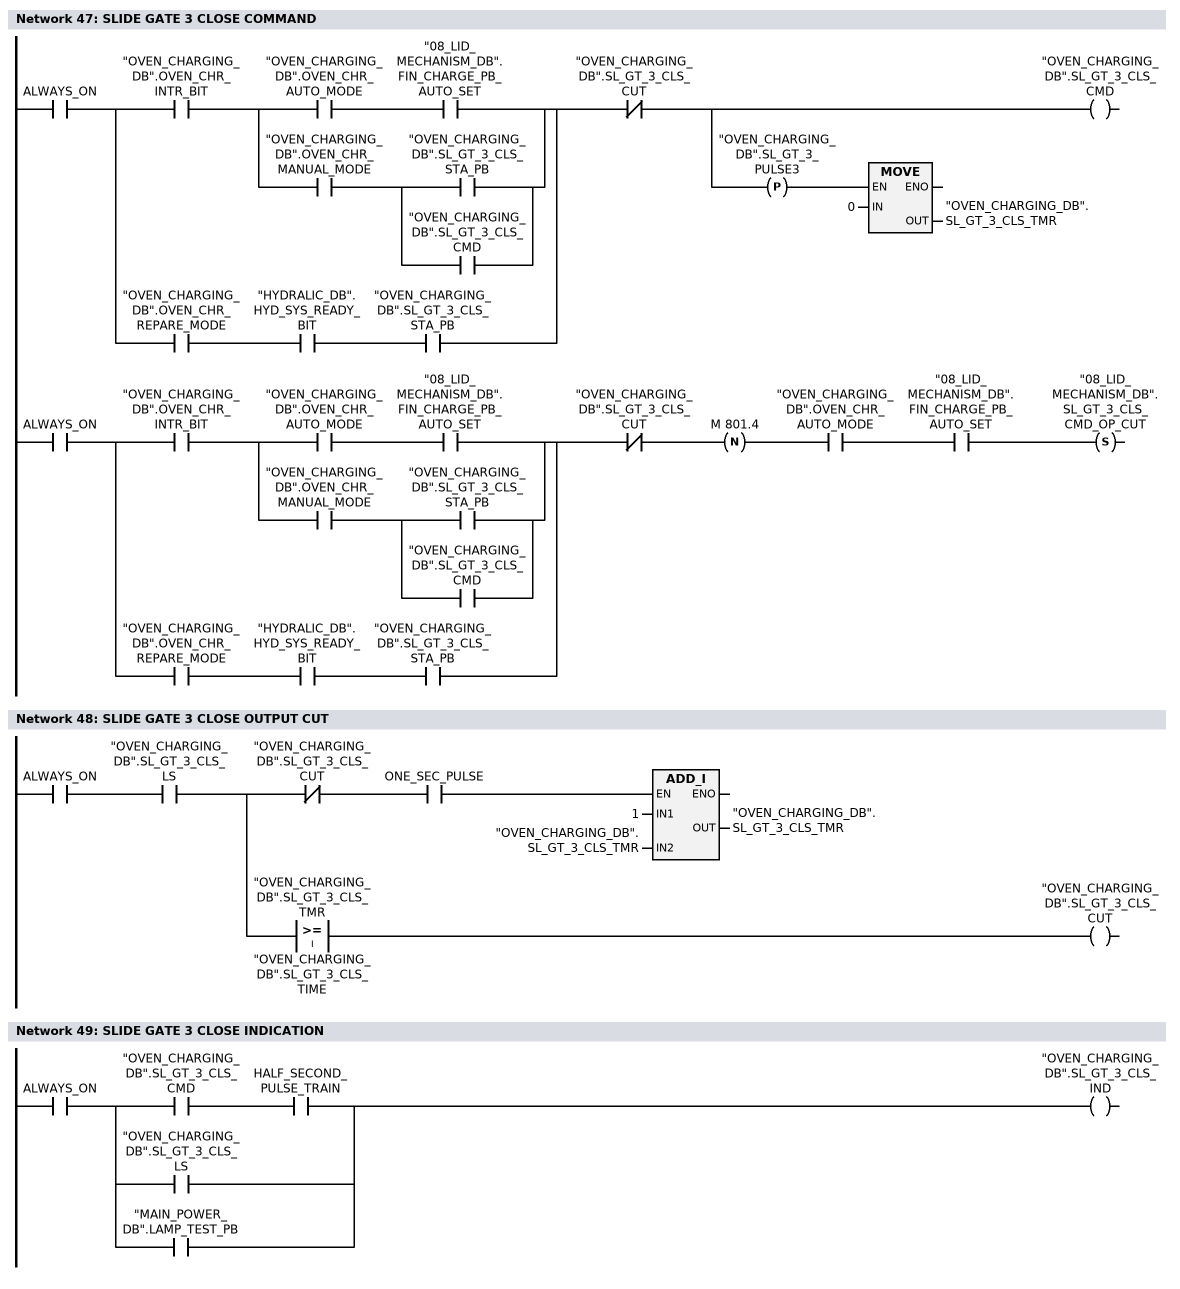
NETWORK
TITLE = SLIDE GATE 3 CLOSE COMMAND
      A     "ALWAYS_ON";
      A(;
      A     "OVEN_CHARGING_DB".OVEN_CHR_INTR_BIT;
      A(;
      A     "OVEN_CHARGING_DB".OVEN_CHR_AUTO_MODE;
      A     "08_LID_MECHANISM_DB".FIN_CHARGE_PB_AUTO_SET;
      O;
      A     "OVEN_CHARGING_DB".OVEN_CHR_MANUAL_MODE;
      A(;
      O     "OVEN_CHARGING_DB".SL_GT_3_CLS_STA_PB;
      O     "OVEN_CHARGING_DB".SL_GT_3_CLS_CMD;
      );
      );
      O;
      A     "OVEN_CHARGING_DB".OVEN_CHR_REPARE_MODE;
      A     "HYDRALIC_DB".HYD_SYS_READY_BIT;
      A     "OVEN_CHARGING_DB".SL_GT_3_CLS_STA_PB;
      );
      AN    "OVEN_CHARGING_DB".SL_GT_3_CLS_CUT;
      =     L 0.0;
      A     L 0.0;
      BLD   102;
      =     "OVEN_CHARGING_DB".SL_GT_3_CLS_CMD;
      A     L 0.0;
      FP    "OVEN_CHARGING_DB".SL_GT_3_PULSE3;
      JNB   _02b;
      L     0;
      T     "OVEN_CHARGING_DB".SL_GT_3_CLS_TMR;
_02b: NOP   0;
      A(;
      A     L 0.0;
      FN    M 801.4;
      );
      A     "OVEN_CHARGING_DB".OVEN_CHR_AUTO_MODE;
      A     "08_LID_MECHANISM_DB".FIN_CHARGE_PB_AUTO_SET;
      S     "08_LID_MECHANISM_DB".SL_GT_3_CLS_CMD_OP_CUT;
NETWORK
TITLE = SLIDE GATE 3 CLOSE OUTPUT CUT
      A     "ALWAYS_ON";
      A     "OVEN_CHARGING_DB".SL_GT_3_CLS_LS;
      =     L 0.0;
      A     L 0.0;
      AN    "OVEN_CHARGING_DB".SL_GT_3_CLS_CUT;
      A     "ONE_SEC_PULSE";
      JNB   _02c;
      L     1;
      L     "OVEN_CHARGING_DB".SL_GT_3_CLS_TMR;
      +I;
      T     "OVEN_CHARGING_DB".SL_GT_3_CLS_TMR;
_02c: NOP   0;
      A     L 0.0;
      A(;
      L     "OVEN_CHARGING_DB".SL_GT_3_CLS_TMR;
      L     "OVEN_CHARGING_DB".SL_GT_3_CLS_TIME;
      >=I;
      );
      =     "OVEN_CHARGING_DB".SL_GT_3_CLS_CUT;
NETWORK
TITLE = SLIDE GATE 3 CLOSE INDICATION
      A     "ALWAYS_ON";
      A(;
      A     "OVEN_CHARGING_DB".SL_GT_3_CLS_CMD;
      A     "HALF_SECOND_PULSE_TRAIN";
      O     "OVEN_CHARGING_DB".SL_GT_3_CLS_LS;
      O     "MAIN_POWER_DB".LAMP_TEST_PB;
      );
      =     "OVEN_CHARGING_DB".SL_GT_3_CLS_IND;
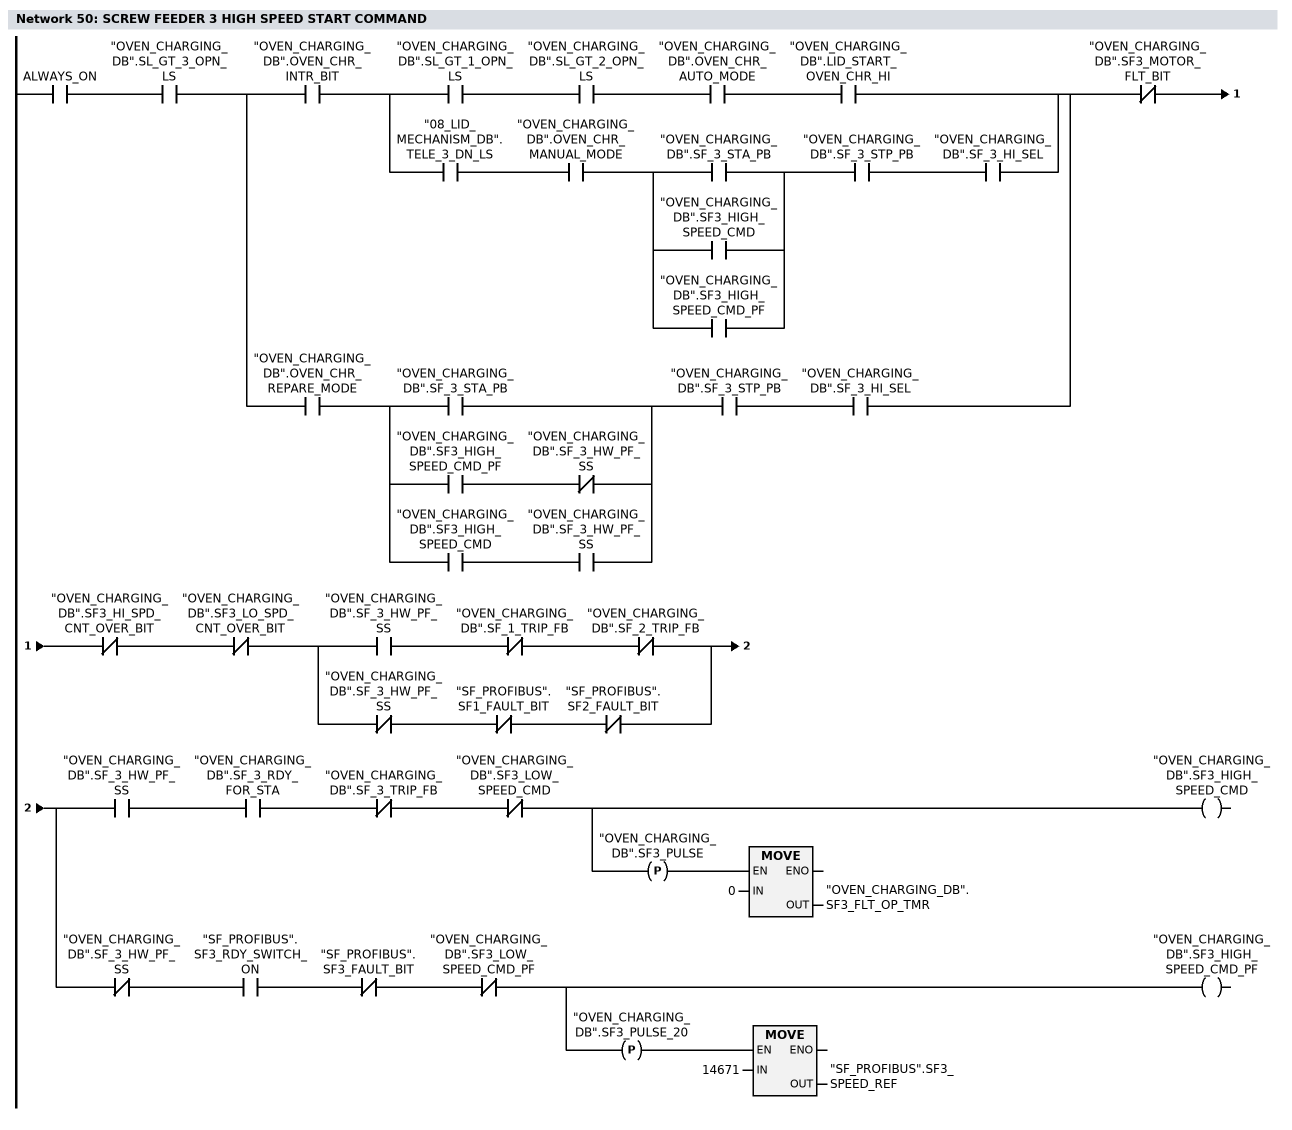
NETWORK
TITLE = SCREW FEEDER 3 HIGH SPEED START COMMAND
      A     "ALWAYS_ON";
      A     "OVEN_CHARGING_DB".SL_GT_3_OPN_LS;
      A(;
      A     "OVEN_CHARGING_DB".OVEN_CHR_INTR_BIT;
      A(;
      A     "OVEN_CHARGING_DB".SL_GT_1_OPN_LS;
      A     "OVEN_CHARGING_DB".SL_GT_2_OPN_LS;
      A     "OVEN_CHARGING_DB".OVEN_CHR_AUTO_MODE;
      A     "OVEN_CHARGING_DB".LID_START_OVEN_CHR_HI;
      O;
      A     "08_LID_MECHANISM_DB".TELE_3_DN_LS;
      A     "OVEN_CHARGING_DB".OVEN_CHR_MANUAL_MODE;
      A(;
      O     "OVEN_CHARGING_DB".SF_3_STA_PB;
      O     "OVEN_CHARGING_DB".SF3_HIGH_SPEED_CMD;
      O     "OVEN_CHARGING_DB".SF3_HIGH_SPEED_CMD_PF;
      );
      A     "OVEN_CHARGING_DB".SF_3_STP_PB;
      A     "OVEN_CHARGING_DB".SF_3_HI_SEL;
      );
      O;
      A     "OVEN_CHARGING_DB".OVEN_CHR_REPARE_MODE;
      A(;
      O     "OVEN_CHARGING_DB".SF_3_STA_PB;
      O;
      A     "OVEN_CHARGING_DB".SF3_HIGH_SPEED_CMD_PF;
      AN    "OVEN_CHARGING_DB".SF_3_HW_PF_SS;
      O;
      A     "OVEN_CHARGING_DB".SF3_HIGH_SPEED_CMD;
      A     "OVEN_CHARGING_DB".SF_3_HW_PF_SS;
      );
      A     "OVEN_CHARGING_DB".SF_3_STP_PB;
      A     "OVEN_CHARGING_DB".SF_3_HI_SEL;
      );
      AN    "OVEN_CHARGING_DB".SF3_MOTOR_FLT_BIT;
      AN    "OVEN_CHARGING_DB".SF3_HI_SPD_CNT_OVER_BIT;
      AN    "OVEN_CHARGING_DB".SF3_LO_SPD_CNT_OVER_BIT;
      A(;
      A     "OVEN_CHARGING_DB".SF_3_HW_PF_SS;
      AN    "OVEN_CHARGING_DB".SF_1_TRIP_FB;
      AN    "OVEN_CHARGING_DB".SF_2_TRIP_FB;
      O;
      AN    "OVEN_CHARGING_DB".SF_3_HW_PF_SS;
      AN    "SF_PROFIBUS".SF1_FAULT_BIT;
      AN    "SF_PROFIBUS".SF2_FAULT_BIT;
      );
      =     L 0.0;
      A     L 0.0;
      A     "OVEN_CHARGING_DB".SF_3_HW_PF_SS;
      A     "OVEN_CHARGING_DB".SF_3_RDY_FOR_STA;
      AN    "OVEN_CHARGING_DB".SF_3_TRIP_FB;
      AN    "OVEN_CHARGING_DB".SF3_LOW_SPEED_CMD;
      =     L 0.1;
      A     L 0.1;
      BLD   102;
      =     "OVEN_CHARGING_DB".SF3_HIGH_SPEED_CMD;
      A     L 0.1;
      FP    "OVEN_CHARGING_DB".SF3_PULSE;
      JNB   _02d;
      L     0;
      T     "OVEN_CHARGING_DB".SF3_FLT_OP_TMR;
_02d: NOP   0;
      A     L 0.0;
      AN    "OVEN_CHARGING_DB".SF_3_HW_PF_SS;
      A     "SF_PROFIBUS".SF3_RDY_SWITCH_ON;
      AN    "SF_PROFIBUS".SF3_FAULT_BIT;
      AN    "OVEN_CHARGING_DB".SF3_LOW_SPEED_CMD_PF;
      =     L 0.1;
      A     L 0.1;
      BLD   102;
      =     "OVEN_CHARGING_DB".SF3_HIGH_SPEED_CMD_PF;
      A     L 0.1;
      FP    "OVEN_CHARGING_DB".SF3_PULSE_20;
      JNB   _02e;
      L     14671;
      T     "SF_PROFIBUS".SF3_SPEED_REF;
_02e: NOP   0;
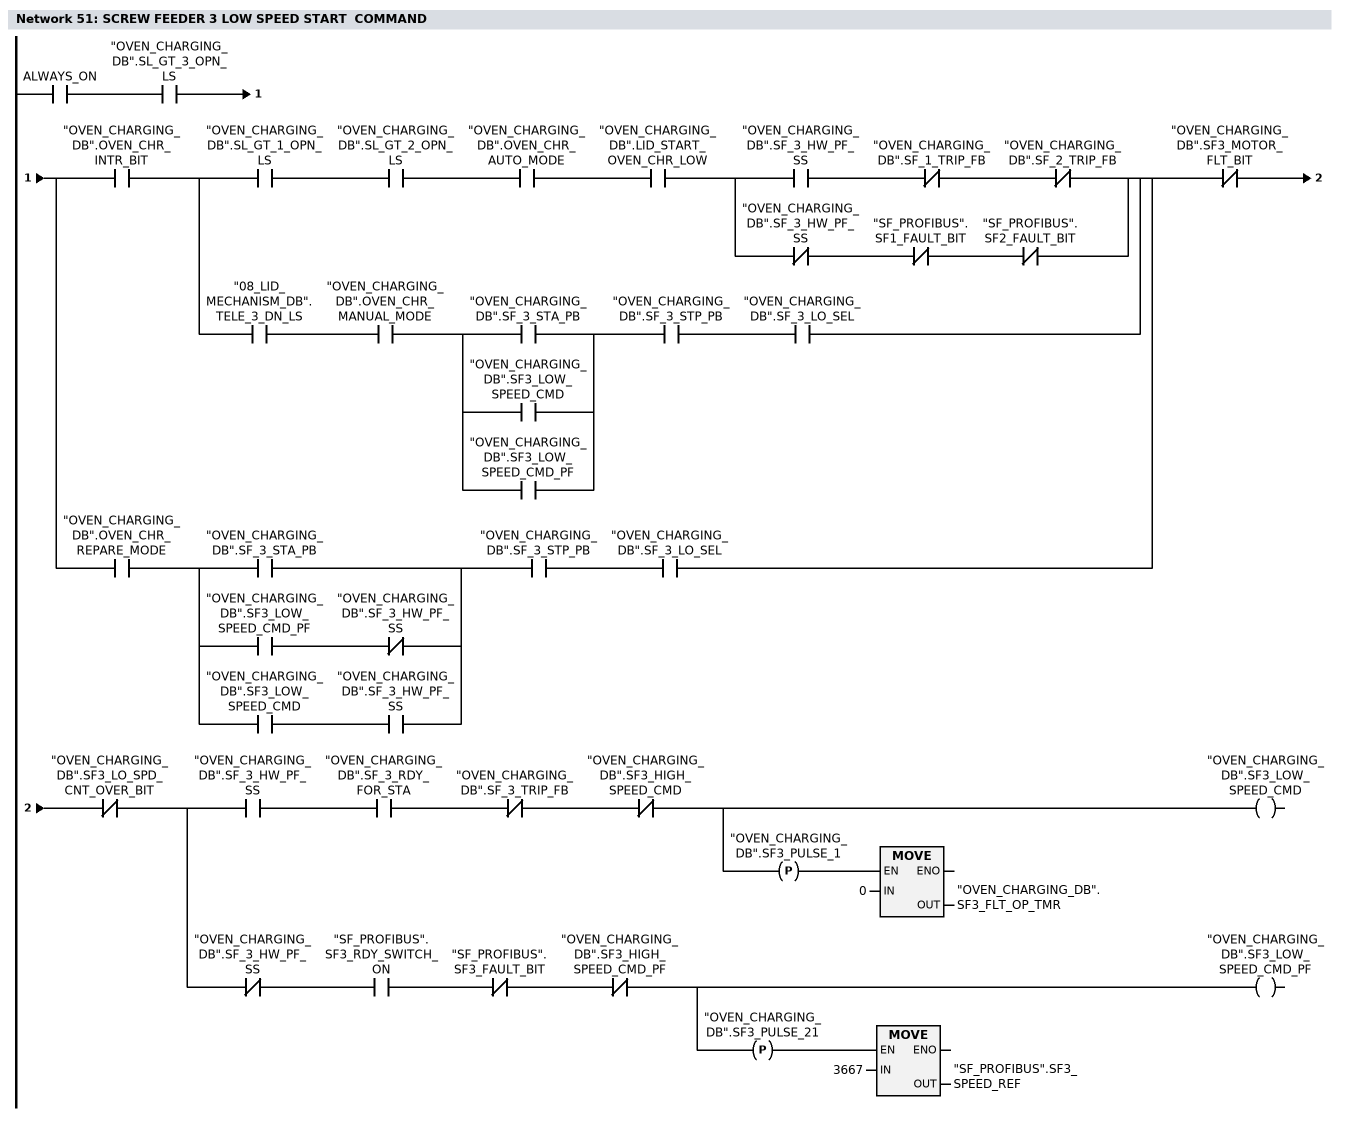
NETWORK
TITLE = SCREW FEEDER 3 LOW SPEED START  COMMAND
      A     "ALWAYS_ON";
      A     "OVEN_CHARGING_DB".SL_GT_3_OPN_LS;
      A(;
      A     "OVEN_CHARGING_DB".OVEN_CHR_INTR_BIT;
      A(;
      A     "OVEN_CHARGING_DB".SL_GT_1_OPN_LS;
      A     "OVEN_CHARGING_DB".SL_GT_2_OPN_LS;
      A     "OVEN_CHARGING_DB".OVEN_CHR_AUTO_MODE;
      A     "OVEN_CHARGING_DB".LID_START_OVEN_CHR_LOW;
      A(;
      A     "OVEN_CHARGING_DB".SF_3_HW_PF_SS;
      AN    "OVEN_CHARGING_DB".SF_1_TRIP_FB;
      AN    "OVEN_CHARGING_DB".SF_2_TRIP_FB;
      O;
      AN    "OVEN_CHARGING_DB".SF_3_HW_PF_SS;
      AN    "SF_PROFIBUS".SF1_FAULT_BIT;
      AN    "SF_PROFIBUS".SF2_FAULT_BIT;
      );
      O;
      A     "08_LID_MECHANISM_DB".TELE_3_DN_LS;
      A     "OVEN_CHARGING_DB".OVEN_CHR_MANUAL_MODE;
      A(;
      O     "OVEN_CHARGING_DB".SF_3_STA_PB;
      O     "OVEN_CHARGING_DB".SF3_LOW_SPEED_CMD;
      O     "OVEN_CHARGING_DB".SF3_LOW_SPEED_CMD_PF;
      );
      A     "OVEN_CHARGING_DB".SF_3_STP_PB;
      A     "OVEN_CHARGING_DB".SF_3_LO_SEL;
      );
      O;
      A     "OVEN_CHARGING_DB".OVEN_CHR_REPARE_MODE;
      A(;
      O     "OVEN_CHARGING_DB".SF_3_STA_PB;
      O;
      A     "OVEN_CHARGING_DB".SF3_LOW_SPEED_CMD_PF;
      AN    "OVEN_CHARGING_DB".SF_3_HW_PF_SS;
      O;
      A     "OVEN_CHARGING_DB".SF3_LOW_SPEED_CMD;
      A     "OVEN_CHARGING_DB".SF_3_HW_PF_SS;
      );
      A     "OVEN_CHARGING_DB".SF_3_STP_PB;
      A     "OVEN_CHARGING_DB".SF_3_LO_SEL;
      );
      AN    "OVEN_CHARGING_DB".SF3_MOTOR_FLT_BIT;
      AN    "OVEN_CHARGING_DB".SF3_LO_SPD_CNT_OVER_BIT;
      =     L 0.0;
      A     L 0.0;
      A     "OVEN_CHARGING_DB".SF_3_HW_PF_SS;
      A     "OVEN_CHARGING_DB".SF_3_RDY_FOR_STA;
      AN    "OVEN_CHARGING_DB".SF_3_TRIP_FB;
      AN    "OVEN_CHARGING_DB".SF3_HIGH_SPEED_CMD;
      =     L 0.1;
      A     L 0.1;
      BLD   102;
      =     "OVEN_CHARGING_DB".SF3_LOW_SPEED_CMD;
      A     L 0.1;
      FP    "OVEN_CHARGING_DB".SF3_PULSE_1;
      JNB   _02f;
      L     0;
      T     "OVEN_CHARGING_DB".SF3_FLT_OP_TMR;
_02f: NOP   0;
      A     L 0.0;
      AN    "OVEN_CHARGING_DB".SF_3_HW_PF_SS;
      A     "SF_PROFIBUS".SF3_RDY_SWITCH_ON;
      AN    "SF_PROFIBUS".SF3_FAULT_BIT;
      AN    "OVEN_CHARGING_DB".SF3_HIGH_SPEED_CMD_PF;
      =     L 0.1;
      A     L 0.1;
      BLD   102;
      =     "OVEN_CHARGING_DB".SF3_LOW_SPEED_CMD_PF;
      A     L 0.1;
      FP    "OVEN_CHARGING_DB".SF3_PULSE_21;
      JNB   _030;
      L     3667;
      T     "SF_PROFIBUS".SF3_SPEED_REF;
_030: NOP   0;
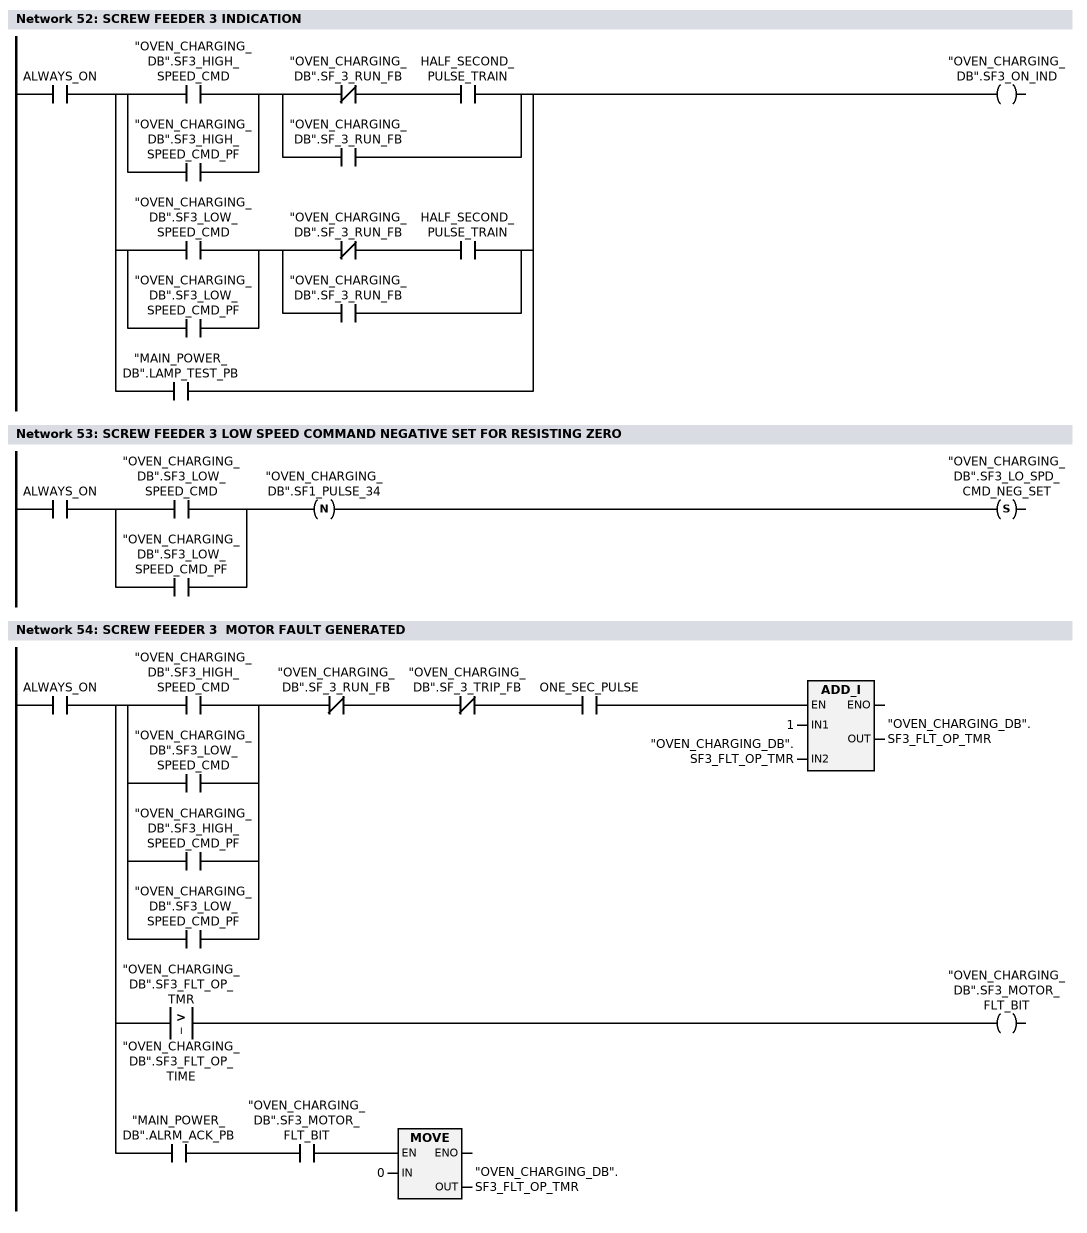
NETWORK
TITLE = SCREW FEEDER 3 INDICATION
      A     "ALWAYS_ON";
      A(;
      A(;
      O     "OVEN_CHARGING_DB".SF3_HIGH_SPEED_CMD;
      O     "OVEN_CHARGING_DB".SF3_HIGH_SPEED_CMD_PF;
      );
      A(;
      AN    "OVEN_CHARGING_DB".SF_3_RUN_FB;
      A     "HALF_SECOND_PULSE_TRAIN";
      O     "OVEN_CHARGING_DB".SF_3_RUN_FB;
      );
      O;
      A(;
      O     "OVEN_CHARGING_DB".SF3_LOW_SPEED_CMD;
      O     "OVEN_CHARGING_DB".SF3_LOW_SPEED_CMD_PF;
      );
      A(;
      AN    "OVEN_CHARGING_DB".SF_3_RUN_FB;
      A     "HALF_SECOND_PULSE_TRAIN";
      O     "OVEN_CHARGING_DB".SF_3_RUN_FB;
      );
      O     "MAIN_POWER_DB".LAMP_TEST_PB;
      );
      =     "OVEN_CHARGING_DB".SF3_ON_IND;
NETWORK
TITLE = SCREW FEEDER 3 LOW SPEED COMMAND NEGATIVE SET FOR RESISTING ZERO
      A     "ALWAYS_ON";
      A(;
      O     "OVEN_CHARGING_DB".SF3_LOW_SPEED_CMD;
      O     "OVEN_CHARGING_DB".SF3_LOW_SPEED_CMD_PF;
      );
      FN    "OVEN_CHARGING_DB".SF1_PULSE_34;
      S     "OVEN_CHARGING_DB".SF3_LO_SPD_CMD_NEG_SET;
NETWORK
TITLE = SCREW FEEDER 3  MOTOR FAULT GENERATED
      A     "ALWAYS_ON";
      =     L 0.0;
      A     L 0.0;
      A(;
      O     "OVEN_CHARGING_DB".SF3_HIGH_SPEED_CMD;
      O     "OVEN_CHARGING_DB".SF3_LOW_SPEED_CMD;
      O     "OVEN_CHARGING_DB".SF3_HIGH_SPEED_CMD_PF;
      O     "OVEN_CHARGING_DB".SF3_LOW_SPEED_CMD_PF;
      );
      AN    "OVEN_CHARGING_DB".SF_3_RUN_FB;
      AN    "OVEN_CHARGING_DB".SF_3_TRIP_FB;
      A     "ONE_SEC_PULSE";
      JNB   _031;
      L     1;
      L     "OVEN_CHARGING_DB".SF3_FLT_OP_TMR;
      +I;
      T     "OVEN_CHARGING_DB".SF3_FLT_OP_TMR;
_031: NOP   0;
      A     L 0.0;
      A(;
      L     "OVEN_CHARGING_DB".SF3_FLT_OP_TMR;
      L     "OVEN_CHARGING_DB".SF3_FLT_OP_TIME;
      >I;
      );
      =     "OVEN_CHARGING_DB".SF3_MOTOR_FLT_BIT;
      A     L 0.0;
      A     "MAIN_POWER_DB".ALRM_ACK_PB;
      A     "OVEN_CHARGING_DB".SF3_MOTOR_FLT_BIT;
      JNB   _032;
      L     0;
      T     "OVEN_CHARGING_DB".SF3_FLT_OP_TMR;
_032: NOP   0;
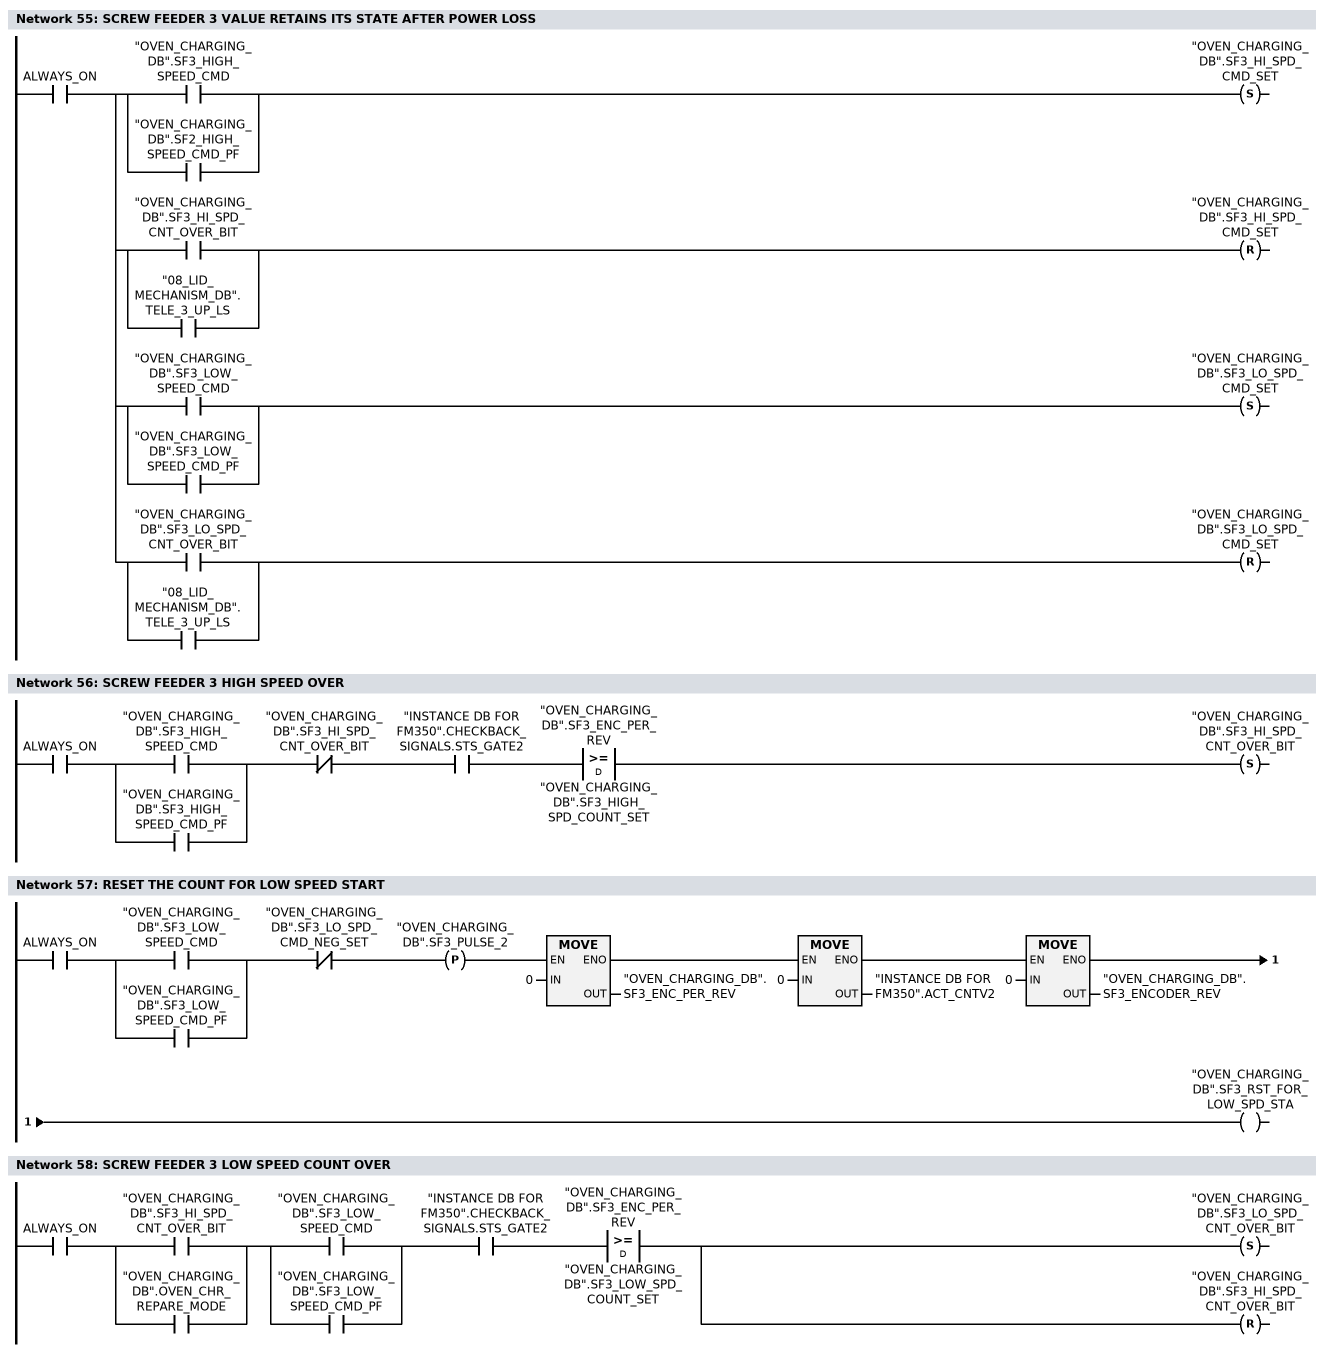
NETWORK
TITLE = SCREW FEEDER 3 VALUE RETAINS ITS STATE AFTER POWER LOSS
      A     "ALWAYS_ON";
      =     L 0.0;
      A     L 0.0;
      A(;
      O     "OVEN_CHARGING_DB".SF3_HIGH_SPEED_CMD;
      O     "OVEN_CHARGING_DB".SF2_HIGH_SPEED_CMD_PF;
      );
      S     "OVEN_CHARGING_DB".SF3_HI_SPD_CMD_SET;
      A     L 0.0;
      A(;
      O     "OVEN_CHARGING_DB".SF3_HI_SPD_CNT_OVER_BIT;
      O     "08_LID_MECHANISM_DB".TELE_3_UP_LS;
      );
      R     "OVEN_CHARGING_DB".SF3_HI_SPD_CMD_SET;
      A     L 0.0;
      A(;
      O     "OVEN_CHARGING_DB".SF3_LOW_SPEED_CMD;
      O     "OVEN_CHARGING_DB".SF3_LOW_SPEED_CMD_PF;
      );
      S     "OVEN_CHARGING_DB".SF3_LO_SPD_CMD_SET;
      A     L 0.0;
      A(;
      O     "OVEN_CHARGING_DB".SF3_LO_SPD_CNT_OVER_BIT;
      O     "08_LID_MECHANISM_DB".TELE_3_UP_LS;
      );
      R     "OVEN_CHARGING_DB".SF3_LO_SPD_CMD_SET;
NETWORK
TITLE = SCREW FEEDER 3 HIGH SPEED OVER
      A     "ALWAYS_ON";
      A(;
      O     "OVEN_CHARGING_DB".SF3_HIGH_SPEED_CMD;
      O     "OVEN_CHARGING_DB".SF3_HIGH_SPEED_CMD_PF;
      );
      AN    "OVEN_CHARGING_DB".SF3_HI_SPD_CNT_OVER_BIT;
      A     "INSTANCE DB FOR FM350".CHECKBACK_SIGNALS.STS_GATE2;
      A(;
      L     "OVEN_CHARGING_DB".SF3_ENC_PER_REV;
      L     "OVEN_CHARGING_DB".SF3_HIGH_SPD_COUNT_SET;
      >=D;
      );
      S     "OVEN_CHARGING_DB".SF3_HI_SPD_CNT_OVER_BIT;
NETWORK
TITLE = RESET THE COUNT FOR LOW SPEED START
      A(;
      A(;
      A     "ALWAYS_ON";
      A(;
      O     "OVEN_CHARGING_DB".SF3_LOW_SPEED_CMD;
      O     "OVEN_CHARGING_DB".SF3_LOW_SPEED_CMD_PF;
      );
      AN    "OVEN_CHARGING_DB".SF3_LO_SPD_CMD_NEG_SET;
      FP    "OVEN_CHARGING_DB".SF3_PULSE_2;
      JNB   _033;
      L     0;
      T     "OVEN_CHARGING_DB".SF3_ENC_PER_REV;
      SET;
      SAVE;
      CLR;
_033: A     BR;
      );
      JNB   _034;
      L     0;
      T     "INSTANCE DB FOR FM350".ACT_CNTV2;
      SET;
      SAVE;
      CLR;
_034: A     BR;
      );
      JNB   _035;
      L     0;
      T     "OVEN_CHARGING_DB".SF3_ENCODER_REV;
      SET;
      SAVE;
      CLR;
_035: A     BR;
      =     "OVEN_CHARGING_DB".SF3_RST_FOR_LOW_SPD_STA;
NETWORK
TITLE = SCREW FEEDER 3 LOW SPEED COUNT OVER
      A     "ALWAYS_ON";
      A(;
      O     "OVEN_CHARGING_DB".SF3_HI_SPD_CNT_OVER_BIT;
      O     "OVEN_CHARGING_DB".OVEN_CHR_REPARE_MODE;
      );
      A(;
      O     "OVEN_CHARGING_DB".SF3_LOW_SPEED_CMD;
      O     "OVEN_CHARGING_DB".SF3_LOW_SPEED_CMD_PF;
      );
      A     "INSTANCE DB FOR FM350".CHECKBACK_SIGNALS.STS_GATE2;
      A(;
      L     "OVEN_CHARGING_DB".SF3_ENC_PER_REV;
      L     "OVEN_CHARGING_DB".SF3_LOW_SPD_COUNT_SET;
      >=D;
      );
      S     "OVEN_CHARGING_DB".SF3_LO_SPD_CNT_OVER_BIT;
      R     "OVEN_CHARGING_DB".SF3_HI_SPD_CNT_OVER_BIT;
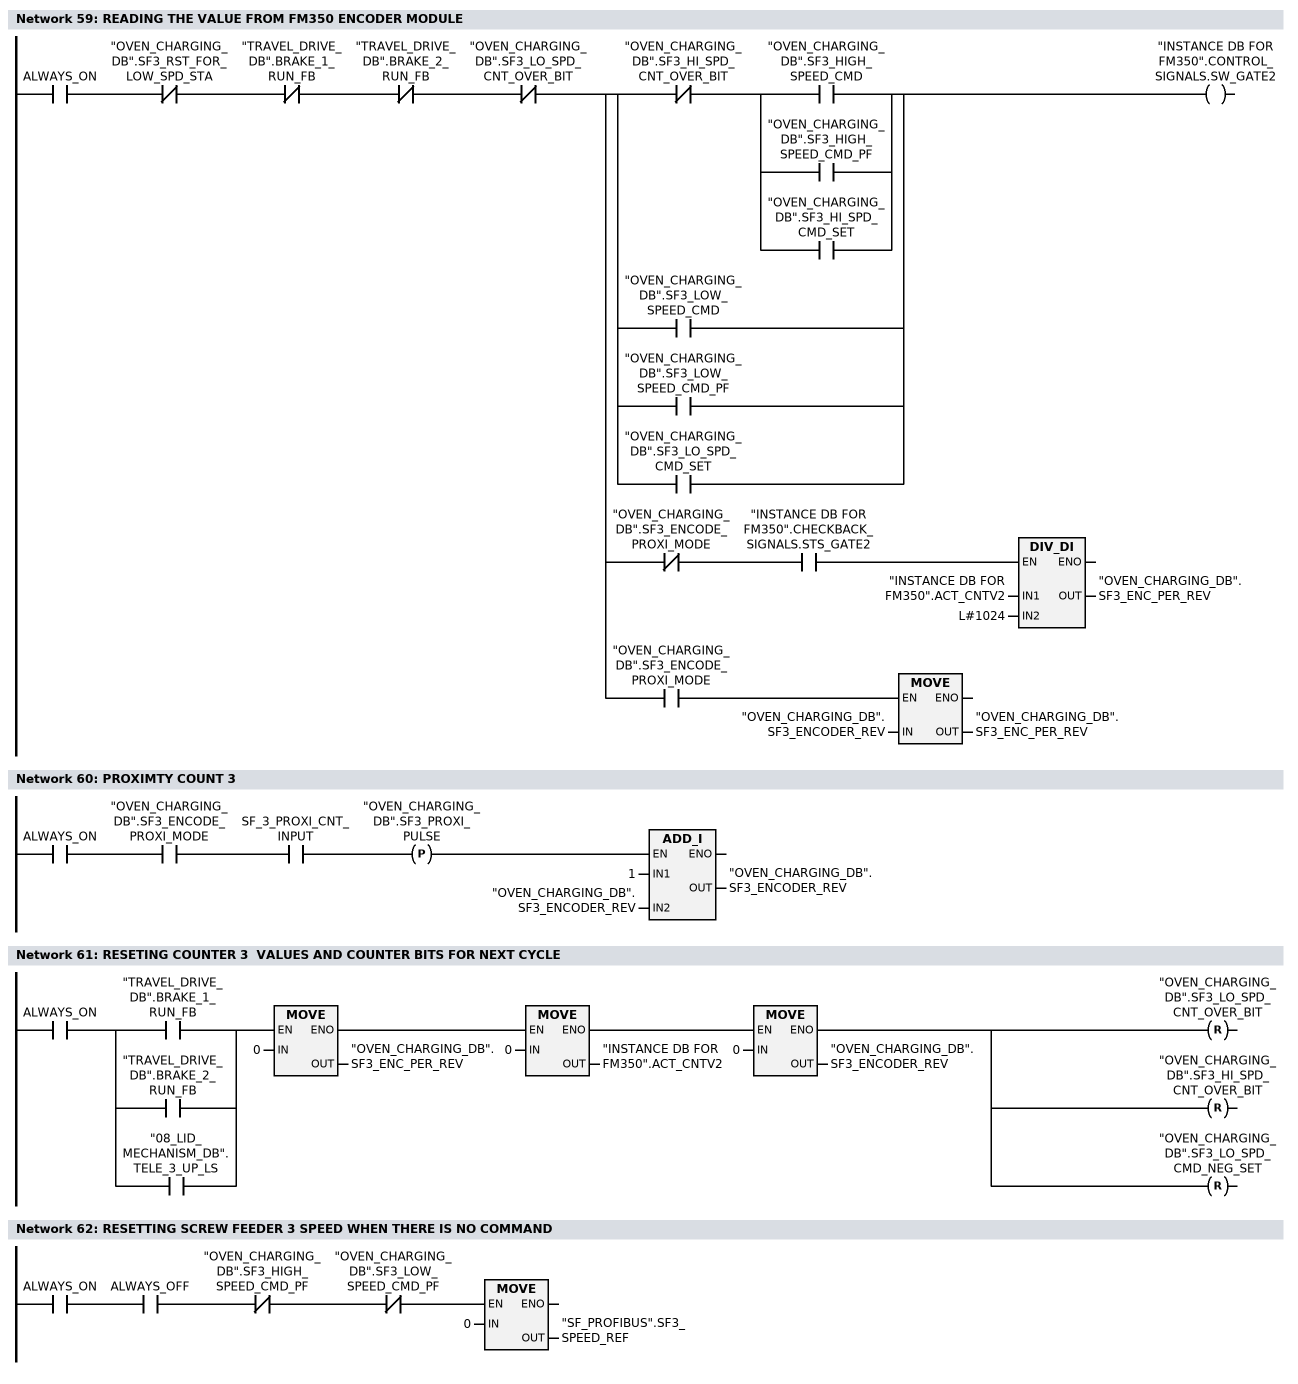
NETWORK
TITLE = READING THE VALUE FROM FM350 ENCODER MODULE 
//FOR FIRST SCREW FEEDER 
      A     "ALWAYS_ON";
      AN    "OVEN_CHARGING_DB".SF3_RST_FOR_LOW_SPD_STA;
      AN    "TRAVEL_DRIVE_DB".BRAKE_1_RUN_FB;
      AN    "TRAVEL_DRIVE_DB".BRAKE_2_RUN_FB;
      AN    "OVEN_CHARGING_DB".SF3_LO_SPD_CNT_OVER_BIT;
      =     L 0.0;
      A     L 0.0;
      A(;
      AN    "OVEN_CHARGING_DB".SF3_HI_SPD_CNT_OVER_BIT;
      A(;
      O     "OVEN_CHARGING_DB".SF3_HIGH_SPEED_CMD;
      O     "OVEN_CHARGING_DB".SF3_HIGH_SPEED_CMD_PF;
      O     "OVEN_CHARGING_DB".SF3_HI_SPD_CMD_SET;
      );
      O     "OVEN_CHARGING_DB".SF3_LOW_SPEED_CMD;
      O     "OVEN_CHARGING_DB".SF3_LOW_SPEED_CMD_PF;
      O     "OVEN_CHARGING_DB".SF3_LO_SPD_CMD_SET;
      );
      =     "INSTANCE DB FOR FM350".CONTROL_SIGNALS.SW_GATE2;
      A     L 0.0;
      AN    "OVEN_CHARGING_DB".SF3_ENCODE_PROXI_MODE;
      A     "INSTANCE DB FOR FM350".CHECKBACK_SIGNALS.STS_GATE2;
      JNB   _036;
      L     "INSTANCE DB FOR FM350".ACT_CNTV2;
      L     L#1024;
      /D;
      T     "OVEN_CHARGING_DB".SF3_ENC_PER_REV;
_036: NOP   0;
      A     L 0.0;
      A     "OVEN_CHARGING_DB".SF3_ENCODE_PROXI_MODE;
      JNB   _037;
      L     "OVEN_CHARGING_DB".SF3_ENCODER_REV;
      T     "OVEN_CHARGING_DB".SF3_ENC_PER_REV;
_037: NOP   0;
NETWORK
TITLE = PROXIMTY COUNT 3
      A     "ALWAYS_ON";
      A     "OVEN_CHARGING_DB".SF3_ENCODE_PROXI_MODE;
      A     "SF_3_PROXI_CNT_INPUT";
      FP    "OVEN_CHARGING_DB".SF3_PROXI_PULSE;
      JNB   _038;
      L     1;
      L     "OVEN_CHARGING_DB".SF3_ENCODER_REV;
      +I;
      T     "OVEN_CHARGING_DB".SF3_ENCODER_REV;
_038: NOP   0;
NETWORK
TITLE = RESETING COUNTER 3  VALUES AND COUNTER BITS FOR NEXT CYCLE
      A(;
      A(;
      A     "ALWAYS_ON";
      A(;
      O     "TRAVEL_DRIVE_DB".BRAKE_1_RUN_FB;
      O     "TRAVEL_DRIVE_DB".BRAKE_2_RUN_FB;
      O     "08_LID_MECHANISM_DB".TELE_3_UP_LS;
      );
      JNB   _039;
      L     0;
      T     "OVEN_CHARGING_DB".SF3_ENC_PER_REV;
      SET;
      SAVE;
      CLR;
_039: A     BR;
      );
      JNB   _03a;
      L     0;
      T     "INSTANCE DB FOR FM350".ACT_CNTV2;
      SET;
      SAVE;
      CLR;
_03a: A     BR;
      );
      JNB   _03b;
      L     0;
      T     "OVEN_CHARGING_DB".SF3_ENCODER_REV;
      SET;
      SAVE;
      CLR;
_03b: A     BR;
      R     "OVEN_CHARGING_DB".SF3_LO_SPD_CNT_OVER_BIT;
      R     "OVEN_CHARGING_DB".SF3_HI_SPD_CNT_OVER_BIT;
      R     "OVEN_CHARGING_DB".SF3_LO_SPD_CMD_NEG_SET;
NETWORK
TITLE = RESETTING SCREW FEEDER 3 SPEED WHEN THERE IS NO COMMAND
      A     "ALWAYS_ON";
      A     "ALWAYS_OFF";
      AN    "OVEN_CHARGING_DB".SF3_HIGH_SPEED_CMD_PF;
      AN    "OVEN_CHARGING_DB".SF3_LOW_SPEED_CMD_PF;
      JNB   _03c;
      L     0;
      T     "SF_PROFIBUS".SF3_SPEED_REF;
_03c: NOP   0;
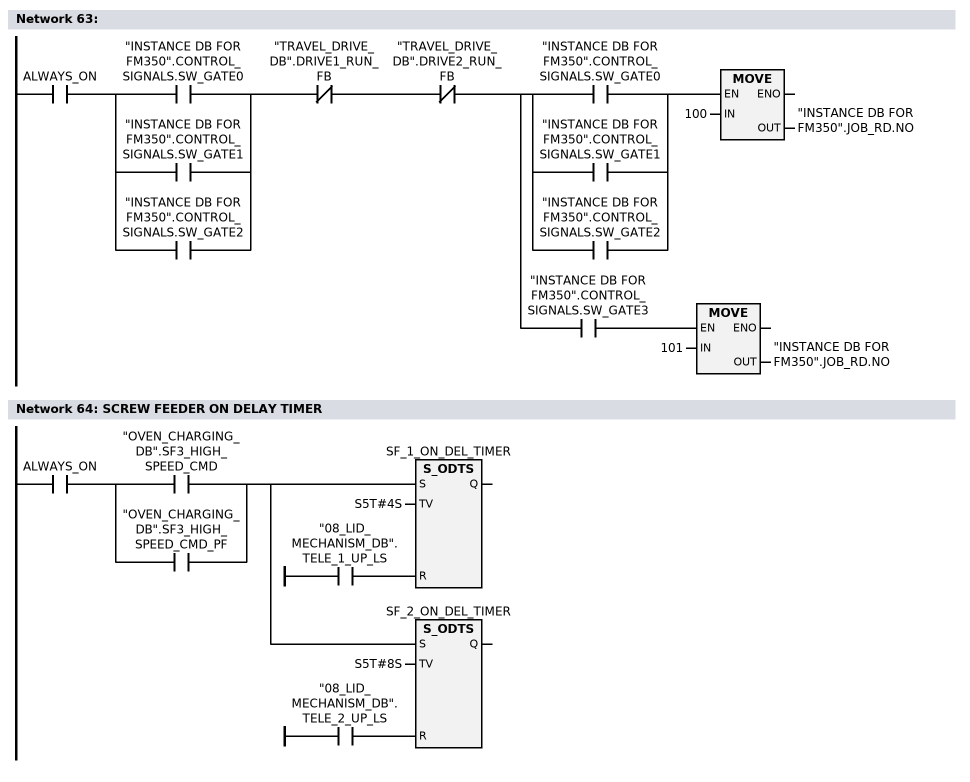
NETWORK
TITLE =
      A     "ALWAYS_ON";
      A(;
      O     "INSTANCE DB FOR FM350".CONTROL_SIGNALS.SW_GATE0;
      O     "INSTANCE DB FOR FM350".CONTROL_SIGNALS.SW_GATE1;
      O     "INSTANCE DB FOR FM350".CONTROL_SIGNALS.SW_GATE2;
      );
      AN    "TRAVEL_DRIVE_DB".DRIVE1_RUN_FB;
      AN    "TRAVEL_DRIVE_DB".DRIVE2_RUN_FB;
      =     L 0.0;
      A     L 0.0;
      A(;
      O     "INSTANCE DB FOR FM350".CONTROL_SIGNALS.SW_GATE0;
      O     "INSTANCE DB FOR FM350".CONTROL_SIGNALS.SW_GATE1;
      O     "INSTANCE DB FOR FM350".CONTROL_SIGNALS.SW_GATE2;
      );
      JNB   _03d;
      L     100;
      T     "INSTANCE DB FOR FM350".JOB_RD.NO;
_03d: NOP   0;
      A     L 0.0;
      A     "INSTANCE DB FOR FM350".CONTROL_SIGNALS.SW_GATE3;
      JNB   _03e;
      L     101;
      T     "INSTANCE DB FOR FM350".JOB_RD.NO;
_03e: NOP   0;
NETWORK
TITLE = SCREW FEEDER ON DELAY TIMER
      A     "ALWAYS_ON";
      A(;
      O     "OVEN_CHARGING_DB".SF3_HIGH_SPEED_CMD;
      O     "OVEN_CHARGING_DB".SF3_HIGH_SPEED_CMD_PF;
      );
      =     L 0.0;
      A     L 0.0;
      L     S5T#4S;
      SS    "SF_1_ON_DEL_TIMER";
      A     "08_LID_MECHANISM_DB".TELE_1_UP_LS;
      R     "SF_1_ON_DEL_TIMER";
      NOP   0;
      NOP   0;
      NOP   0;
      A     L 0.0;
      L     S5T#8S;
      SS    "SF_2_ON_DEL_TIMER";
      A     "08_LID_MECHANISM_DB".TELE_2_UP_LS;
      R     "SF_2_ON_DEL_TIMER";
      NOP   0;
      NOP   0;
      NOP   0;
END_FUNCTION

FUNCTION "LID_1_MECHANISM" : VOID	// FC 11
//AUTO SEQ
//Prepare to charge pb 
//Carriage Fwd 
//Vert Down 
//Mag On
//Osc On
//3s 
//Osc off
//Lid at mag
//Ver Up
//Car Ret 
//// Frm clnr down if bypass
//Car fwd 
//car Ver cln pos down 
//Frm clnr Mtr on 
//5s 
//off 
//car Ver  up 
//Car Ret //
//Teles Down 
AUTHOR : Arun
VERSION : 0.1
BEGIN
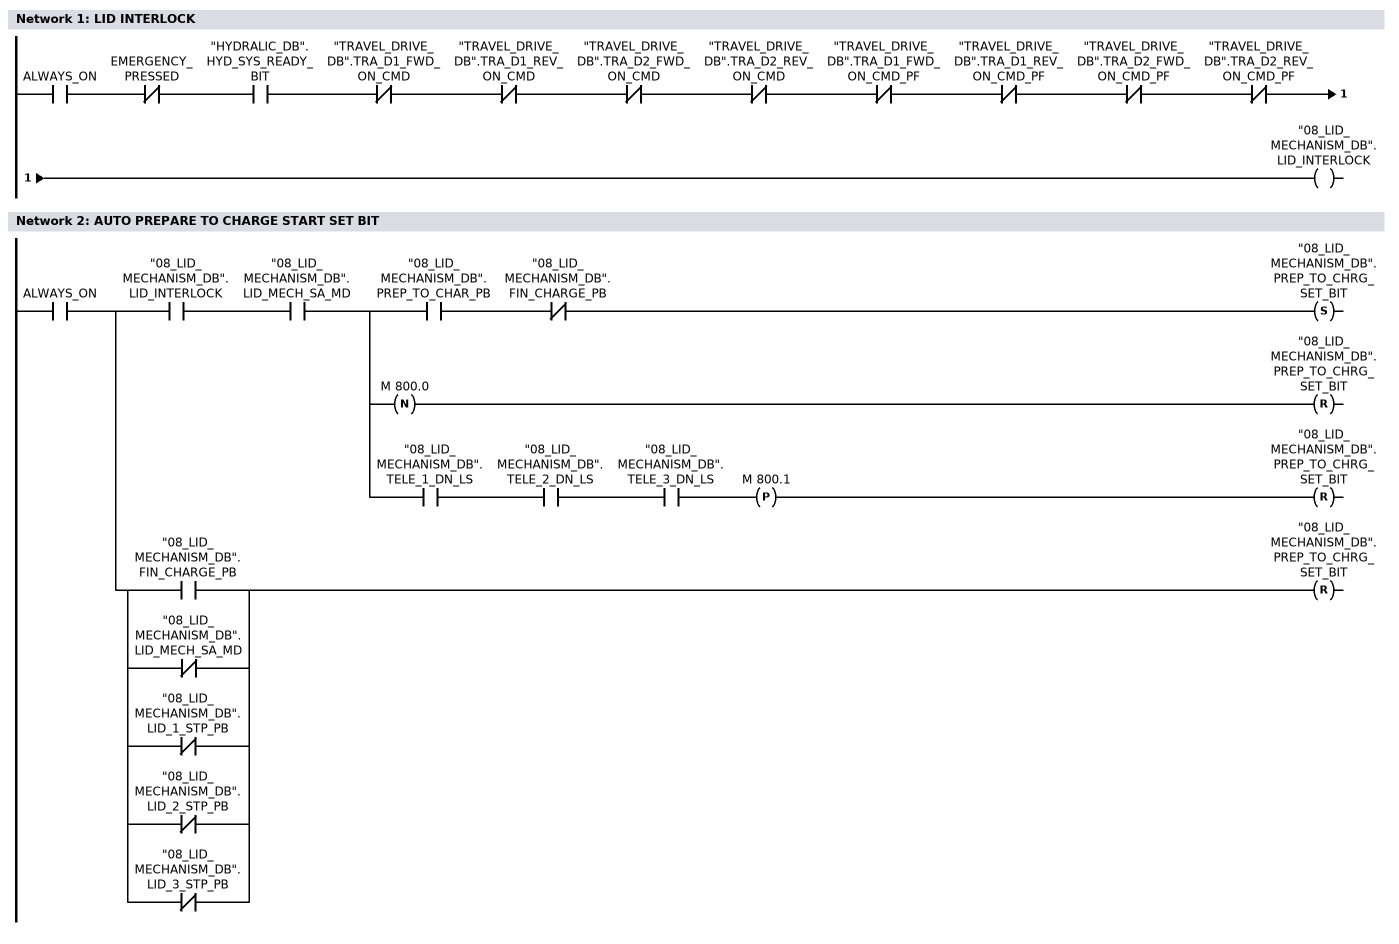
NETWORK
TITLE = LID INTERLOCK
      A     "ALWAYS_ON";
      AN    "EMERGENCY_PRESSED";
      A     "HYDRALIC_DB".HYD_SYS_READY_BIT;
      AN    "TRAVEL_DRIVE_DB".TRA_D1_FWD_ON_CMD;
      AN    "TRAVEL_DRIVE_DB".TRA_D1_REV_ON_CMD;
      AN    "TRAVEL_DRIVE_DB".TRA_D2_FWD_ON_CMD;
      AN    "TRAVEL_DRIVE_DB".TRA_D2_REV_ON_CMD;
      AN    "TRAVEL_DRIVE_DB".TRA_D1_FWD_ON_CMD_PF;
      AN    "TRAVEL_DRIVE_DB".TRA_D1_REV_ON_CMD_PF;
      AN    "TRAVEL_DRIVE_DB".TRA_D2_FWD_ON_CMD_PF;
      AN    "TRAVEL_DRIVE_DB".TRA_D2_REV_ON_CMD_PF;
      =     "08_LID_MECHANISM_DB".LID_INTERLOCK;
NETWORK
TITLE = AUTO PREPARE TO CHARGE START SET BIT 
      A     "ALWAYS_ON";
      =     L 0.0;
      A     L 0.0;
      A     "08_LID_MECHANISM_DB".LID_INTERLOCK;
      A     "08_LID_MECHANISM_DB".LID_MECH_SA_MD;
      =     L 0.1;
      A     L 0.1;
      A     "08_LID_MECHANISM_DB".PREP_TO_CHAR_PB;
      AN    "08_LID_MECHANISM_DB".FIN_CHARGE_PB;
      S     "08_LID_MECHANISM_DB".PREP_TO_CHRG_SET_BIT;
      A     L 0.1;
      FN    M 800.0;
      R     "08_LID_MECHANISM_DB".PREP_TO_CHRG_SET_BIT;
      A     L 0.1;
      A     "08_LID_MECHANISM_DB".TELE_1_DN_LS;
      A     "08_LID_MECHANISM_DB".TELE_2_DN_LS;
      A     "08_LID_MECHANISM_DB".TELE_3_DN_LS;
      FP    M 800.1;
      R     "08_LID_MECHANISM_DB".PREP_TO_CHRG_SET_BIT;
      A     L 0.0;
      A(;
      O     "08_LID_MECHANISM_DB".FIN_CHARGE_PB;
      ON    "08_LID_MECHANISM_DB".LID_MECH_SA_MD;
      ON    "08_LID_MECHANISM_DB".LID_1_STP_PB;
      ON    "08_LID_MECHANISM_DB".LID_2_STP_PB;
      ON    "08_LID_MECHANISM_DB".LID_3_STP_PB;
      );
      R     "08_LID_MECHANISM_DB".PREP_TO_CHRG_SET_BIT;
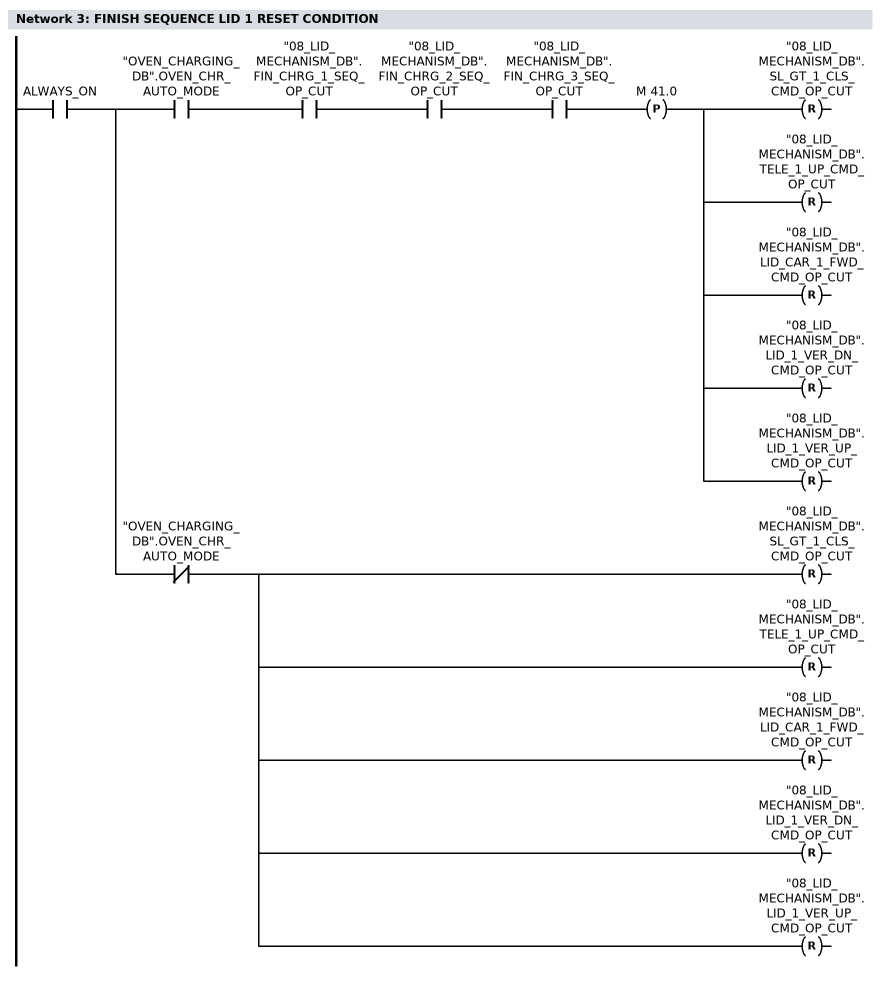
NETWORK
TITLE = FINISH SEQUENCE LID 1 RESET CONDITION
      A     "ALWAYS_ON";
      =     L 0.0;
      A     L 0.0;
      A     "OVEN_CHARGING_DB".OVEN_CHR_AUTO_MODE;
      A     "08_LID_MECHANISM_DB".FIN_CHRG_1_SEQ_OP_CUT;
      A     "08_LID_MECHANISM_DB".FIN_CHRG_2_SEQ_OP_CUT;
      A     "08_LID_MECHANISM_DB".FIN_CHRG_3_SEQ_OP_CUT;
      FP    M 41.0;
      R     "08_LID_MECHANISM_DB".SL_GT_1_CLS_CMD_OP_CUT;
      R     "08_LID_MECHANISM_DB".TELE_1_UP_CMD_OP_CUT;
      R     "08_LID_MECHANISM_DB".LID_CAR_1_FWD_CMD_OP_CUT;
      R     "08_LID_MECHANISM_DB".LID_1_VER_DN_CMD_OP_CUT;
      R     "08_LID_MECHANISM_DB".LID_1_VER_UP_CMD_OP_CUT;
      A     L 0.0;
      AN    "OVEN_CHARGING_DB".OVEN_CHR_AUTO_MODE;
      R     "08_LID_MECHANISM_DB".SL_GT_1_CLS_CMD_OP_CUT;
      R     "08_LID_MECHANISM_DB".TELE_1_UP_CMD_OP_CUT;
      R     "08_LID_MECHANISM_DB".LID_CAR_1_FWD_CMD_OP_CUT;
      R     "08_LID_MECHANISM_DB".LID_1_VER_DN_CMD_OP_CUT;
      R     "08_LID_MECHANISM_DB".LID_1_VER_UP_CMD_OP_CUT;
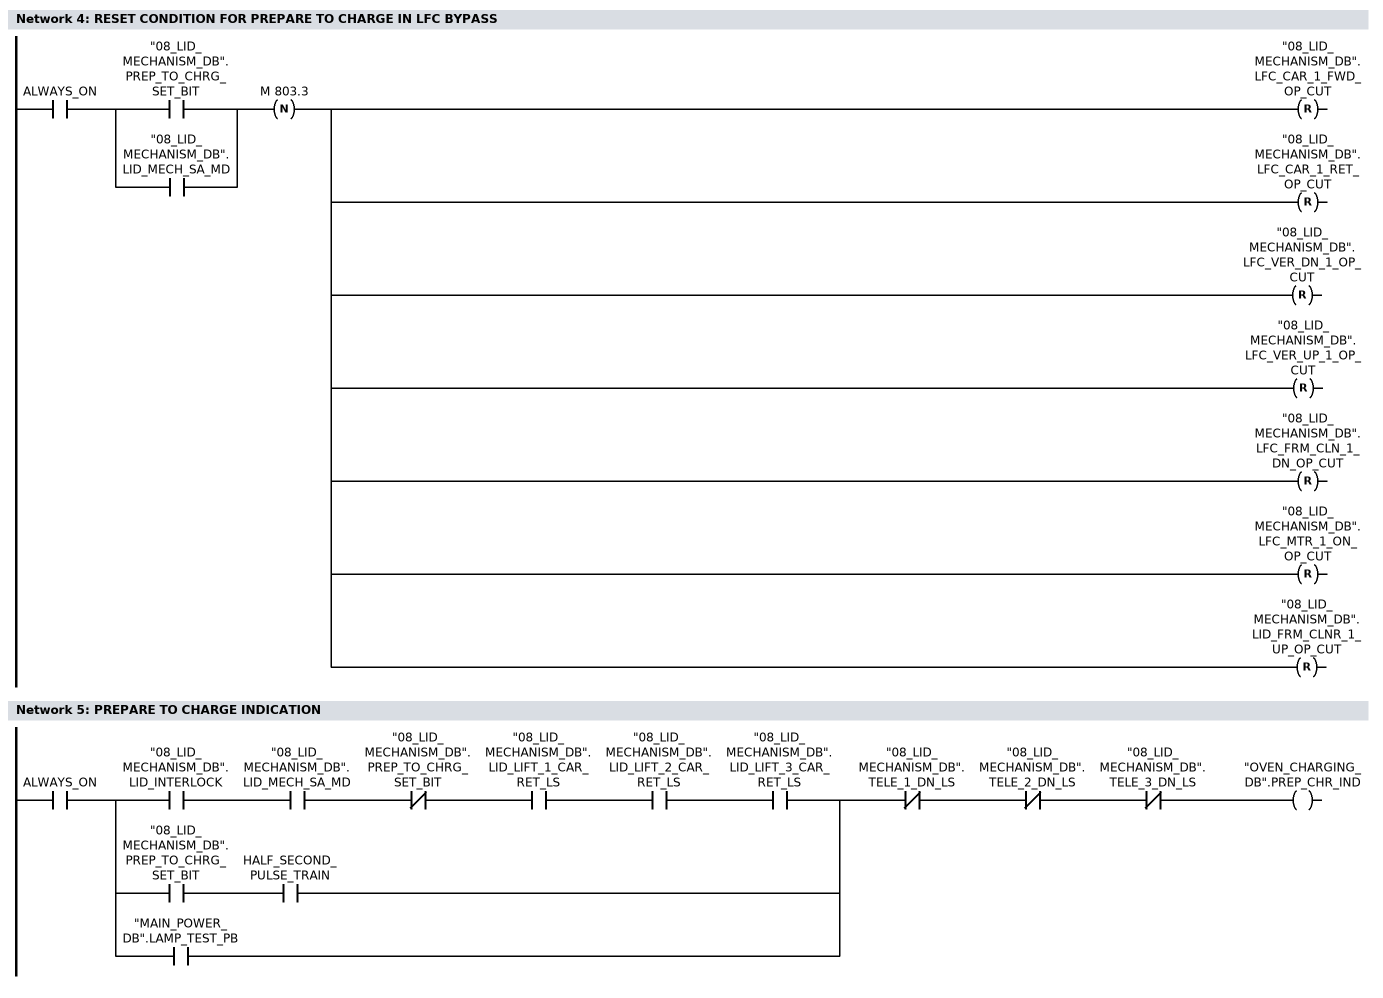
NETWORK
TITLE = RESET CONDITION FOR PREPARE TO CHARGE IN LFC BYPASS
      A     "ALWAYS_ON";
      A(;
      O     "08_LID_MECHANISM_DB".PREP_TO_CHRG_SET_BIT;
      O     "08_LID_MECHANISM_DB".LID_MECH_SA_MD;
      );
      FN    M 803.3;
      R     "08_LID_MECHANISM_DB".LFC_CAR_1_FWD_OP_CUT;
      R     "08_LID_MECHANISM_DB".LFC_CAR_1_RET_OP_CUT;
      R     "08_LID_MECHANISM_DB".LFC_VER_DN_1_OP_CUT;
      R     "08_LID_MECHANISM_DB".LFC_VER_UP_1_OP_CUT;
      R     "08_LID_MECHANISM_DB".LFC_FRM_CLN_1_DN_OP_CUT;
      R     "08_LID_MECHANISM_DB".LFC_MTR_1_ON_OP_CUT;
      R     "08_LID_MECHANISM_DB".LID_FRM_CLNR_1_UP_OP_CUT;
NETWORK
TITLE = PREPARE TO CHARGE INDICATION
      A     "ALWAYS_ON";
      A(;
      A     "08_LID_MECHANISM_DB".LID_INTERLOCK;
      A     "08_LID_MECHANISM_DB".LID_MECH_SA_MD;
      AN    "08_LID_MECHANISM_DB".PREP_TO_CHRG_SET_BIT;
      A     "08_LID_MECHANISM_DB".LID_LIFT_1_CAR_RET_LS;
      A     "08_LID_MECHANISM_DB".LID_LIFT_2_CAR_RET_LS;
      A     "08_LID_MECHANISM_DB".LID_LIFT_3_CAR_RET_LS;
      O;
      A     "08_LID_MECHANISM_DB".PREP_TO_CHRG_SET_BIT;
      A     "HALF_SECOND_PULSE_TRAIN";
      O     "MAIN_POWER_DB".LAMP_TEST_PB;
      );
      AN    "08_LID_MECHANISM_DB".TELE_1_DN_LS;
      AN    "08_LID_MECHANISM_DB".TELE_2_DN_LS;
      AN    "08_LID_MECHANISM_DB".TELE_3_DN_LS;
      =     "OVEN_CHARGING_DB".PREP_CHR_IND;
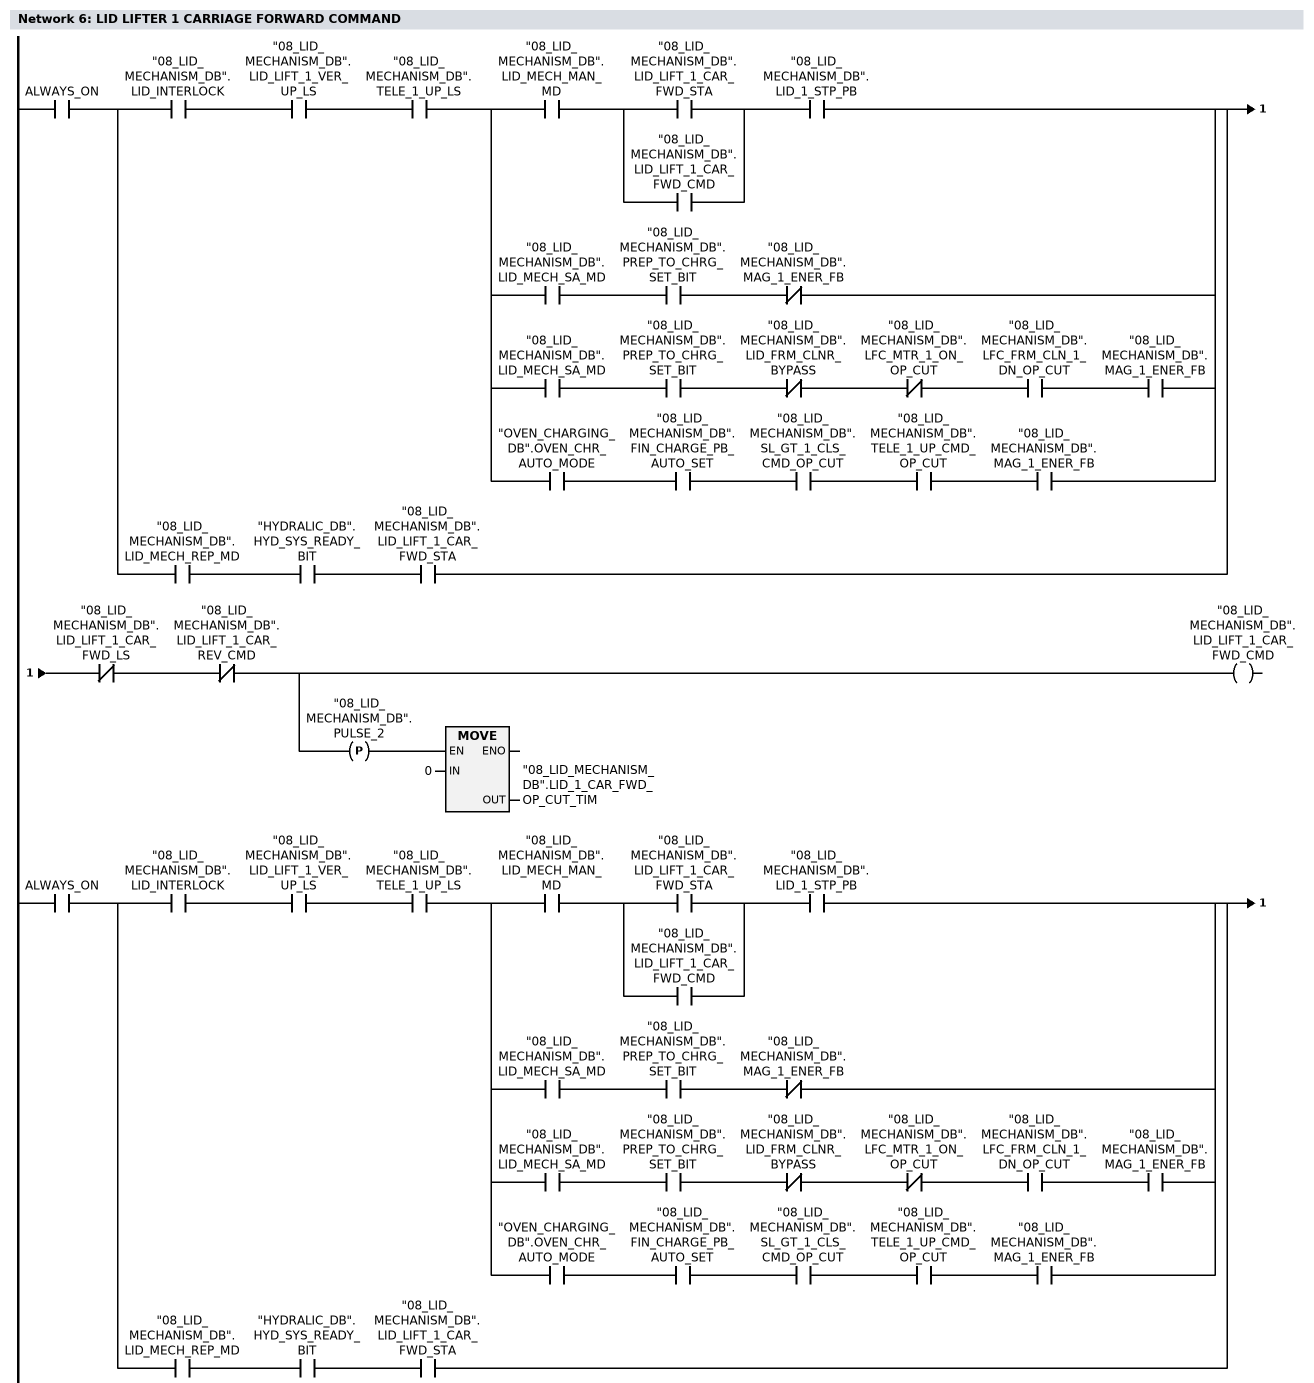
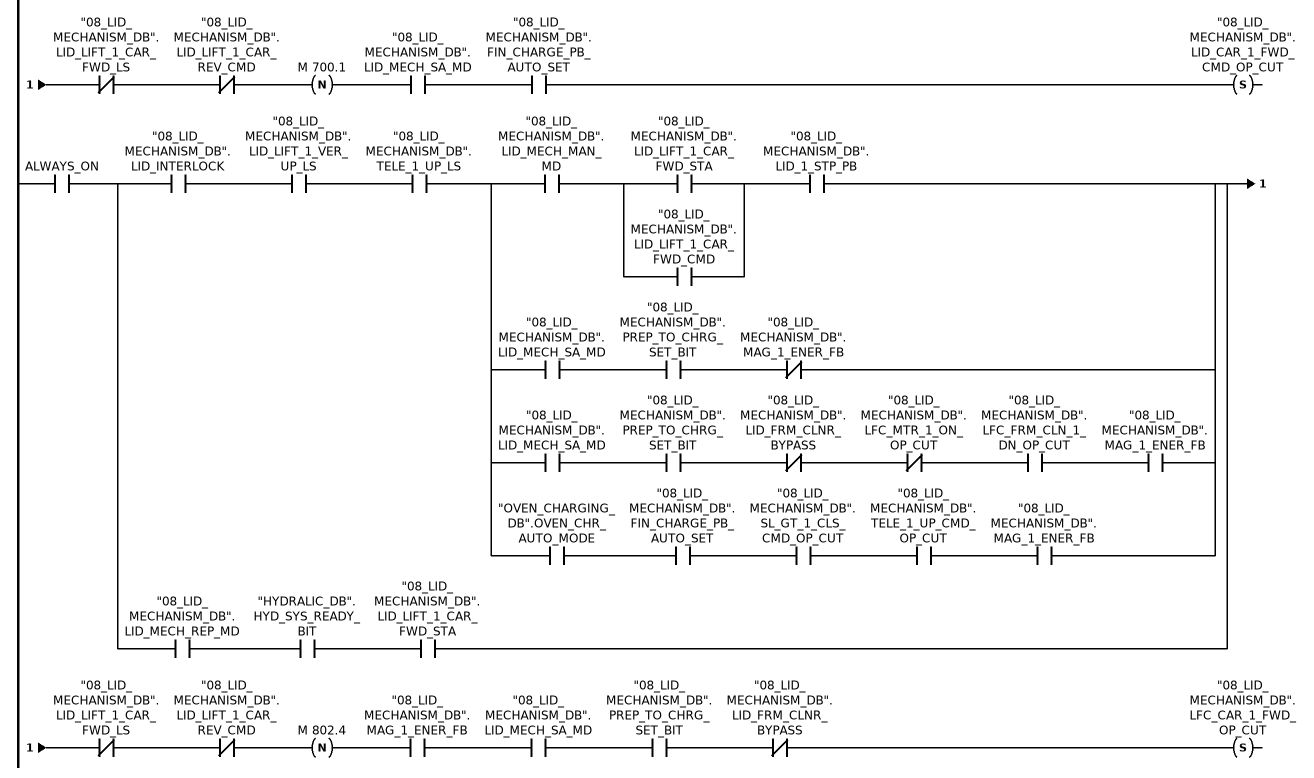
NETWORK
TITLE = LID LIFTER 1 CARRIAGE FORWARD COMMAND
      A     "ALWAYS_ON";
      A(;
      A     "08_LID_MECHANISM_DB".LID_INTERLOCK;
      A     "08_LID_MECHANISM_DB".LID_LIFT_1_VER_UP_LS;
      A     "08_LID_MECHANISM_DB".TELE_1_UP_LS;
      A(;
      A     "08_LID_MECHANISM_DB".LID_MECH_MAN_MD;
      A(;
      O     "08_LID_MECHANISM_DB".LID_LIFT_1_CAR_FWD_STA;
      O     "08_LID_MECHANISM_DB".LID_LIFT_1_CAR_FWD_CMD;
      );
      A     "08_LID_MECHANISM_DB".LID_1_STP_PB;
      O;
      A     "08_LID_MECHANISM_DB".LID_MECH_SA_MD;
      A     "08_LID_MECHANISM_DB".PREP_TO_CHRG_SET_BIT;
      AN    "08_LID_MECHANISM_DB".MAG_1_ENER_FB;
      O;
      A     "08_LID_MECHANISM_DB".LID_MECH_SA_MD;
      A     "08_LID_MECHANISM_DB".PREP_TO_CHRG_SET_BIT;
      AN    "08_LID_MECHANISM_DB".LID_FRM_CLNR_BYPASS;
      AN    "08_LID_MECHANISM_DB".LFC_MTR_1_ON_OP_CUT;
      A     "08_LID_MECHANISM_DB".LFC_FRM_CLN_1_DN_OP_CUT;
      A     "08_LID_MECHANISM_DB".MAG_1_ENER_FB;
      O;
      A     "OVEN_CHARGING_DB".OVEN_CHR_AUTO_MODE;
      A     "08_LID_MECHANISM_DB".FIN_CHARGE_PB_AUTO_SET;
      A     "08_LID_MECHANISM_DB".SL_GT_1_CLS_CMD_OP_CUT;
      A     "08_LID_MECHANISM_DB".TELE_1_UP_CMD_OP_CUT;
      A     "08_LID_MECHANISM_DB".MAG_1_ENER_FB;
      );
      O;
      A     "08_LID_MECHANISM_DB".LID_MECH_REP_MD;
      A     "HYDRALIC_DB".HYD_SYS_READY_BIT;
      A     "08_LID_MECHANISM_DB".LID_LIFT_1_CAR_FWD_STA;
      );
      AN    "08_LID_MECHANISM_DB".LID_LIFT_1_CAR_FWD_LS;
      AN    "08_LID_MECHANISM_DB".LID_LIFT_1_CAR_REV_CMD;
      =     L 0.0;
      A     L 0.0;
      BLD   102;
      =     "08_LID_MECHANISM_DB".LID_LIFT_1_CAR_FWD_CMD;
      A     L 0.0;
      FP    "08_LID_MECHANISM_DB".PULSE_2;
      JNB   _001;
      L     0;
      T     "08_LID_MECHANISM_DB".LID_1_CAR_FWD_OP_CUT_TIM;
_001: NOP   0;
      A(;
      A     L 0.0;
      FN    M 700.1;
      );
      A     "08_LID_MECHANISM_DB".LID_MECH_SA_MD;
      A     "08_LID_MECHANISM_DB".FIN_CHARGE_PB_AUTO_SET;
      S     "08_LID_MECHANISM_DB".LID_CAR_1_FWD_CMD_OP_CUT;
      A(;
      A     L 0.0;
      FN    M 802.4;
      );
      A     "08_LID_MECHANISM_DB".MAG_1_ENER_FB;
      A     "08_LID_MECHANISM_DB".LID_MECH_SA_MD;
      A     "08_LID_MECHANISM_DB".PREP_TO_CHRG_SET_BIT;
      AN    "08_LID_MECHANISM_DB".LID_FRM_CLNR_BYPASS;
      S     "08_LID_MECHANISM_DB".LFC_CAR_1_FWD_OP_CUT;
